      #angle axis calculation
      normal_vector = cross_product(touch1_pose_to_touch2_pose_if_no_rotation, touch1_pose_to_touch2_pose)
      normal_vector_norm = norm(normal_vector)
      if (normal_vector_norm > 10e-6):
        rotation_angle_rad = asin( normal_vector_norm / (norm(touch1_pose_to_touch2_pose_if_no_rotation) * norm(touch1_pose_to_touch2_pose) ) )
        normal_vector_to_angle_axis_multiply_norm_factor = rotation_angle_rad / normal_vector_norm
        angle_axis = [normal_vector[0] * normal_vector_to_angle_axis_multiply_norm_factor, normal_vector[1] * normal_vector_to_angle_axis_multiply_norm_factor, normal_vector[2] * normal_vector_to_angle_axis_multiply_norm_factor]
        rotation_offset_pose = p[0, 0, 0, angle_axis[0], angle_axis[1], angle_axis[2]]

        #rotate touch1 pose using touch2 information
        touch1_pose_rotated = pose_trans(touch1_pose, rotation_offset_pose)
      else:
        touch1_pose_rotated = touch1_pose
      end

      # relocate the feature using touch1_rotated_pose
      return relocate_xyzr(feature_init_pose, touch1_init_pose, touch1_pose_rotated)
    end

    def relocate_1_touch(touch_init_pose, touch_pose, feature_init_pose, feature_actual_pose):
      touch_initial_pose_in_initial_feature_frame = pose_trans(pose_inv(feature_init_pose), touch_init_pose)
      touch_actual_pose_in_actual_feature_frame = pose_trans(pose_inv(feature_actual_pose), touch_pose)

      # difference between touch poses in their respective feature frame
      touch_pose_offset = pose_sub(touch_actual_pose_in_actual_feature_frame, touch_initial_pose_in_initial_feature_frame)

      # remove all rotation from offset
      touch_pose_offset[3] = 0
      touch_pose_offset[4] = 0
      touch_pose_offset[5] = 0

      # apply pose offset to actual feature
      return pose_trans(feature_actual_pose, touch_pose_offset)
    end
    ##############################################
    # PALLETIZER INITIALIZATION
    ##############################################
    if(not palletizerXmlRpcClient.acknowledgePalletStates()):
      checkForScriptPreparationException()
      halt
    end

    ##############################################
    # PALLETIZER-RELATED VARIABLES AND METHODS
    ##############################################
    def rq_is_last_box_of_layer(box_id, end_of_layer_boxes):
      number_of_layers = length(end_of_layer_boxes)
      i = 0
      while i < number_of_layers:
        if box_id == end_of_layer_boxes[i]:
          return True
          break
        end
        i = i + 1
      end
      return False
    end

    def rq_is_palletOne_activated(pallet_one_current_box_count, pallet_two_current_box_count, second_pallet_activated):
      return ((pallet_one_current_box_count == 0) and (pallet_two_current_box_count == 0) and (not second_pallet_activated)) or (pallet_one_current_box_count > pallet_two_current_box_count)
    end
    global servojId = 2
  rq_collision_detection_stop()
  # end: URCap Installation Node
  # begin: URCap Installation Node
  #   Source: Robotiq_Grippers, 1.8.6.7016, Robotiq Inc.
  #   Type: Gripper
  rq_gripper_socket_ip_address = "127.0.0.1"
  rq_gripper_socket_port = 63352

  rq_comm_check_fail_counter = [0, 0, 0, 0]

  rq_read_act = [-1, -1, -1, -1]
  rq_read_gto = [-1, -1, -1, -1]
  rq_read_for = [-1, -1, -1, -1]
  rq_read_spe = [-1, -1, -1, -1]
  rq_read_obj = [-1, -1, -1, -1]
  rq_read_sta = [-1, -1, -1, -1]
  rq_read_flt = [-1, -1, -1, -1]
  rq_read_pos = [-1, -1, -1, -1]
  rq_read_pre = [-1, -1, -1, -1]
  rq_read_lbp = [-1, -1, -1, -1]
  rq_read_lrd = [-1, -1, -1, -1]
  rq_read_lbl = [-1, -1, -1, -1]
  rq_read_lgn = [-1, -1, -1, -1]
  rq_read_msc = [-1, -1, -1, -1]
  rq_read_mod = [-1, -1, -1, -1]
  rq_read_cou = [-1, -1, -1, -1]
  rq_read_ncy = [-1, -1, -1, -1]
  rq_read_dst = [-1, -1, -1, -1]
  rq_read_pco = [-1, -1, -1, -1]

  rq_string_initial_value = "N/A"

  rq_read_snu_1 = rq_string_initial_value
  rq_read_snu_2 = rq_string_initial_value
  rq_read_snu_3 = rq_string_initial_value
  rq_read_snu_4 = rq_string_initial_value

  rq_read_fwv_1 = rq_string_initial_value
  rq_read_fwv_2 = rq_string_initial_value
  rq_read_fwv_3 = rq_string_initial_value
  rq_read_fwv_4 = rq_string_initial_value

  rq_read_ver_1 = rq_string_initial_value
  rq_read_ver_2 = rq_string_initial_value
  rq_read_ver_3 = rq_string_initial_value
  rq_read_ver_4 = rq_string_initial_value

  rq_read_act_req = [True, True, True, True]
  rq_read_gto_req = [True, True, True, True]
  rq_read_for_req = [True, True, True, True]
  rq_read_spe_req = [True, True, True, True]
  rq_read_obj_req = [True, True, True, True]
  rq_read_sta_req = [True, True, True, True]
  rq_read_flt_req = [True, True, True, True]
  rq_read_pos_req = [True, True, True, True]
  rq_read_pre_req = [True, True, True, True]
  rq_read_lbp_req = [True, True, True, True]
  rq_read_lrd_req = [True, True, True, True]
  rq_read_lbl_req = [True, True, True, True]
  rq_read_lgn_req = [True, True, True, True]
  rq_read_msc_req = [True, True, True, True]
  rq_read_mod_req = [True, True, True, True]
  rq_read_cou_req = [True, True, True, True]
  rq_read_ncy_req = [True, True, True, True]
  rq_read_dst_req = [True, True, True, True]
  rq_read_pco_req = [True, True, True, True]

  rq_read_snu_1_req = False
  rq_read_snu_2_req = False
  rq_read_snu_3_req = False
  rq_read_snu_4_req = False

  rq_read_fwv_1_req = False
  rq_read_fwv_2_req = False
  rq_read_fwv_3_req = False
  rq_read_fwv_4_req = False

  rq_read_ver_1_req = False
  rq_read_ver_2_req = False
  rq_read_ver_3_req = False
  rq_read_ver_4_req = False

  rq_write_act_request = [False, False, False, False]
  rq_write_gto_request = [False, False, False, False]
  rq_write_atr_request = [False, False, False, False]
  rq_write_ard_request = [False, False, False, False]
  rq_write_pos_request = [False, False, False, False]
  rq_write_lbp_request = [False, False, False, False]
  rq_write_lrd_request = [False, False, False, False]
  rq_write_lbl_request = [False, False, False, False]
  rq_write_lgn_request = [False, False, False, False]
  rq_write_msc_request = [False, False, False, False]
  rq_write_mod_request = [False, False, False, False]

  rq_write_act = [-1, -1, -1, -1]
  rq_write_gto = [-1, -1, -1, -1]
  rq_write_atr = [-1, -1, -1, -1]
  rq_write_ard = [-1, -1, -1, -1]
  rq_write_for = [-1, -1, -1, -1]
  rq_write_spe = [-1, -1, -1, -1]
  rq_write_pos = [-1, -1, -1, -1]
  rq_write_lbp = [-1, -1, -1, -1]
  rq_write_lrd = [-1, -1, -1, -1]
  rq_write_lbl = [-1, -1, -1, -1]
  rq_write_lgn = [-1, -1, -1, -1]
  rq_write_msc = [-1, -1, -1, -1]
  rq_write_mod = [-1, -1, -1, -1]

  rq_write_act_previous = rq_write_act
  rq_write_gto_previous = rq_write_gto
  rq_write_atr_previous = rq_write_atr
  rq_write_ard_previous = rq_write_ard
  rq_write_for_previous = rq_write_for
  rq_write_spe_previous = rq_write_spe
  rq_write_pos_previous = rq_write_pos
  rq_write_lbp_previous = rq_write_lbp
  rq_write_lrd_previous = rq_write_lrd
  rq_write_lbl_previous = rq_write_lbl
  rq_write_lgn_previous = rq_write_lgn
  rq_write_msc_previous = rq_write_msc
  rq_write_mod_previous = rq_write_mod

  gripper_connected = [False, False, False, False]
  gripper_socket_open = [False, False, False, False]
  rq_comm_clear_socket_buffer_enabled = [True, True, True, True]
  rq_comm_check_counter = 0
  rq_gripper_communication_thread_started = False

  thread rq_gripper_communication():
      rq_comm_read_constants()
      rq_comm_read_variables()
      rq_comm_initialize_write_values()

      while(True):
          rq_comm_clear_socket_buffer()
          rq_comm_check()
          rq_comm_read_variables()
          rq_comm_write_variables()

          rq_gripper_communication_thread_started = True
          sleep(0.008)
      end
  end

  def rq_socket_to_index(gripper_socket="1"):
      # Patch in case gripper_socket is an integer
      gripper_socket_string = str_cat("", gripper_socket)

      if(gripper_socket_string == "1"):
          return 0
      elif(gripper_socket_string == "2"):
          return 1
      elif(gripper_socket_string == "3"):
          return 2
      elif(gripper_socket_string == "4"):
          return 3
      end
      return 0
  end

  def rq_index_to_socket(index=0):
      if(index == 0):
          return "1"
      elif(index == 1):
          return "2"
      elif(index == 2):
          return "3"
      elif(index == 3):
          return "4"
      end
      return "1"
  end

  def rq_comm_check():
      index = 0
      rq_comm_check_fail_counter_max = 99999

      if(rq_comm_check_counter < 50):
          rq_comm_check_counter = rq_comm_check_counter + 1
      else:
          rq_comm_check_counter = 0

          while(index <= 3):
              socket = rq_index_to_socket(index)

              if(gripper_connected[index]):
                  # Patch in case gripper_socket is an integer
                  gripper_socket_string = str_cat("", socket)

                  sid_list = rq_get_sid(socket)
                  is_gripper_in_sid_list = rq_is_gripper_in_sid_list(gripper_socket_string, sid_list)

                  if(is_gripper_in_sid_list):
                      rq_comm_check_fail_counter[index] = 0
                  else:
                      rq_comm_check_fail_counter[index] = rq_comm_check_fail_counter[index] + 1
                  end

                  if(rq_comm_check_fail_counter[index] > rq_comm_check_fail_counter_max):
                      message = str_cat("Communication lost with Robotiq's Gripper Slave ID ", gripper_socket_string)
                      popup(message, "Communication Error", False, True, True)
                  end
              end
              index = index + 1
          end
      end
  end

  def rq_init_comm_if_connected(gripper_sid=9, gripper_socket="1"):
      if(not is_gripper_socket_open(gripper_socket)):
        open_gripper_socket(gripper_socket)
      end

      socket_sid_set = rq_set_sid(gripper_sid, gripper_socket)

      if(socket_sid_set):
          # Patch in case gripper_socket is an integer
          gripper_socket_string = str_cat("", gripper_socket)

          sid_list = rq_get_sid(gripper_socket)
          is_gripper_in_sid_list = rq_is_gripper_in_sid_list(gripper_socket_string, sid_list)

          if(is_gripper_in_sid_list):
              rq_set_gripper_connected(gripper_socket_string)
              return True
          end
      end

      return False
  end

  def open_gripper_socket(gripper_socket="1"):
      is_open = socket_open(rq_gripper_socket_ip_address, rq_gripper_socket_port, gripper_socket)
      set_gripper_socket_open(gripper_socket, is_open)
  end

  def rq_close_gripper_socket(gripper_socket="1"):
      socket_close(gripper_socket)
      set_gripper_socket_open(gripper_socket, False)
      rq_set_gripper_connected(gripper_socket, False)
  end


  def is_gripper_socket_open(gripper_socket="1"):
      return gripper_socket_open[rq_socket_to_index(gripper_socket)]
  end

  def set_gripper_socket_open(gripper_socket, is_open):
      gripper_socket_open[rq_socket_to_index(gripper_socket)] = is_open
  end

  def rq_set_gripper_connected(gripper_socket="1", connected = True):
      gripper_connected[rq_socket_to_index(gripper_socket)] = connected
  end

  def rq_is_gripper_connected(gripper_id="1"):
      return gripper_connected[rq_socket_to_index(gripper_id)]
  end

  def rq_set_sid(gripper_sid=9, gripper_socket="1"):
      socket_set_var("SID", gripper_sid,  gripper_socket)
      ack = socket_read_byte_list(3, gripper_socket)
      return is_ack(ack)
  end

  def rq_get_sid(gripper_socket="1"):
      socket_send_string("GET SID", gripper_socket)
      sid_list = socket_read_byte_list(17, gripper_socket)
      return sid_list
  end

  def rq_wait_for_gripper_connected():
      gripper_socket = "gripper_conn_socket"
      socket_open(rq_gripper_socket_ip_address, rq_gripper_socket_port, gripper_socket)

      remainingRetries = 2000
      sid_list = rq_get_sid(gripper_socket)
      gripper_is_connected = rq_is_any_gripper_connected(sid_list)

      while(not gripper_is_connected and remainingRetries > 0):
          remainingRetries = remainingRetries - 1
          sid_list = rq_get_sid(gripper_socket)
          gripper_is_connected = rq_is_any_gripper_connected(sid_list)
      end

      socket_close(gripper_socket)
  end

  def rq_is_any_gripper_connected(sid_list):
      is_gripper_1_connected = rq_is_gripper1_in_sid_list(sid_list)
      is_gripper_2_connected = rq_is_gripper2_in_sid_list(sid_list)
      is_gripper_3_connected = rq_is_gripper3_in_sid_list(sid_list)
      is_gripper_4_connected = rq_is_gripper4_in_sid_list(sid_list)

      return is_gripper_1_connected or is_gripper_2_connected or is_gripper_3_connected or is_gripper_4_connected
  end

  def rq_is_gripper_ascii_in_sid_list(gripper_ascii_sid, sid_list):
      sid_list_length = sid_list[0]
      sid_list_empty_length = 2

      if (sid_list_length <= sid_list_empty_length):
          return False
      end

      sid1 = sid_list[2]
      sid2 = sid_list[5]
      sid3 = sid_list[8]
      sid4 = sid_list[11]

      return sid1 == gripper_ascii_sid or sid2 == gripper_ascii_sid or sid3 == gripper_ascii_sid or sid4 == gripper_ascii_sid
  end

  def rq_is_gripper_in_sid_list(gripper_socket_string, sid_list):
      if(gripper_socket_string == "1"):
          return rq_is_gripper1_in_sid_list(sid_list)
      elif(gripper_socket_string == "2"):
          return rq_is_gripper2_in_sid_list(sid_list)
      elif(gripper_socket_string == "3"):
          return rq_is_gripper3_in_sid_list(sid_list)
      elif(gripper_socket_string == "4"):
          return rq_is_gripper4_in_sid_list(sid_list)
      end
      return False
  end

  def rq_is_gripper1_in_sid_list(sid_list):
      gripper_1_sid_ascii = 57
      return rq_is_gripper_ascii_in_sid_list(gripper_1_sid_ascii, sid_list)
  end

  def rq_is_gripper2_in_sid_list(sid_list):
      gripper_2_sid_ascii = 50
      return rq_is_gripper_ascii_in_sid_list(gripper_2_sid_ascii, sid_list)
  end

  def rq_is_gripper3_in_sid_list(sid_list):
      gripper_3_sid_ascii = 51
      return rq_is_gripper_ascii_in_sid_list(gripper_3_sid_ascii, sid_list)
  end

  def rq_is_gripper4_in_sid_list(sid_list):
      gripper_4_sid_ascii = 52
      return rq_is_gripper_ascii_in_sid_list(gripper_4_sid_ascii, sid_list)
  end

  def rq_comm_clear_socket_buffer():
      index = 0

      while(index <= 3):
          socket = rq_index_to_socket(index)

          if(gripper_connected[index] and rq_comm_clear_socket_buffer_enabled[index]):
              byte_in_buffer = socket_read_byte_list(1, socket, 0.002)
              while(byte_in_buffer[0] >= 1):
                  byte_in_buffer = socket_read_byte_list(1, socket, 0.002)
              end
              rq_comm_clear_socket_buffer_enabled[index] = False
          end
          index = index + 1
      end
  end

  def rq_comm_initialize_write_values():
      index = 0

      while(index <= 3):
          socket = rq_index_to_socket(index)

          if(gripper_connected[index]):

              if(rq_write_act[index] == -1 and rq_read_act[index] != -1):
                  rq_write_act[index] = rq_read_act[index]
                  rq_write_act_previous[index] = rq_read_act[index]
              elif(rq_write_act_previous[index] == -1 and rq_read_act[index] != -1):
                  rq_write_act_previous[index] = rq_read_act[index]
              end

              if(rq_write_gto[index] == -1 and rq_read_gto[index] != -1):
                  rq_write_gto[index] = rq_read_gto[index]
                  rq_write_gto_previous[index] = rq_read_gto[index]
              elif(rq_write_gto_previous[index] == -1 and rq_read_gto[index] != -1):
                  rq_write_gto_previous[index] = rq_read_gto[index]
              end

              if(rq_write_for[index] == -1 and rq_read_for[index] != -1):
                  rq_write_for[index] = rq_read_for[index]
                  rq_write_for_previous[index] = rq_read_for[index]
              elif(rq_write_for_previous[index] == -1 and rq_read_for[index] != -1):
                  rq_write_for_previous[index] = rq_read_for[index]
              end

              if(rq_write_spe[index] == -1 and rq_read_spe[index] != -1):
                  rq_write_spe[index] = rq_read_spe[index]
                  rq_write_spe_previous[index] = rq_read_spe[index]
              elif(rq_write_spe_previous[index] == -1 and rq_read_spe[index] != -1):
                  rq_write_spe_previous[index] = rq_read_spe[index]
              end

              if(rq_write_pos[index] == -1 and rq_read_pos[index] != -1):
                  rq_write_pos[index] = rq_read_pos[index]
                  rq_write_pos_previous[index] = rq_read_pos[index]
              elif(rq_write_pos_previous[index] == -1 and rq_read_pos[index] != -1):
                  rq_write_pos_previous[index] = rq_read_pos[index]
              end

              if(rq_write_lbp[index] == -1 and rq_read_lbp[index] != -1):
                  rq_write_lbp[index] = rq_read_lbp[index]
                  rq_write_lbp_previous[index] = rq_read_lbp[index]
              elif(rq_write_lbp_previous[index] == -1 and rq_read_lbp[index] != -1):
                  rq_write_lbp_previous[index] = rq_read_lbp[index]
              end

              if(rq_write_lrd[index] == -1 and rq_read_lrd[index] != -1):
                  rq_write_lrd[index] = rq_read_lrd[index]
                  rq_write_lrd_previous[index] = rq_read_lrd[index]
              elif(rq_write_lrd_previous[index] == -1 and rq_read_lrd[index] != -1):
                  rq_write_lrd_previous[index] = rq_read_lrd[index]
              end

              if(rq_write_lbl[index] == -1 and rq_read_lbl[index] != -1):
                  rq_write_lbl[index] = rq_read_lbl[index]
                  rq_write_lbl_previous[index] = rq_read_lbl[index]
              elif(rq_write_lbl_previous[index] == -1 and rq_read_lbl[index] != -1):
                  rq_write_lbl_previous[index] = rq_read_lbl[index]
              end

              if(rq_write_lgn[index] == -1 and rq_read_lgn[index] != -1):
                  rq_write_lgn[index] = rq_read_lgn[index]
                  rq_write_lgn_previous[index] = rq_read_lgn[index]
              elif(rq_write_lgn_previous[index] == -1 and rq_read_lgn[index] != -1):
                  rq_write_lgn_previous[index] = rq_read_lgn[index]
              end

              if(rq_write_msc[index] == -1 and rq_read_msc[index] != -1):
                  rq_write_msc[index] = rq_read_msc[index]
                  rq_write_msc_previous[index] = rq_read_msc[index]
              elif(rq_write_msc_previous[index] == -1 and rq_read_msc[index] != -1):
                  rq_write_msc_previous[index] = rq_read_msc[index]
              end

              if(rq_write_mod[index] == -1 and rq_read_mod[index] != -1):
                  rq_write_mod[index] = rq_read_mod[index]
                  rq_write_mod_previous[index] = rq_read_mod[index]
              elif(rq_write_mod_previous[index] == -1 and rq_read_mod[index] != -1):
                  rq_write_mod_previous[index] = rq_read_mod[index]
              end

          end
          index = index + 1
      end
  end

  def rq_comm_set_var(var, value=0, gripper_socket="1"):
      socket_set_var(var, value, gripper_socket)
      return socket_read_byte_list(3, gripper_socket)
  end

  def rq_comm_set_pos_spe_for(pos=0, speed=0, force=0, gripper_socket="1"):
      socket_send_string("SET POS", gripper_socket)
      socket_send_byte(32, gripper_socket)
      socket_send_string(pos, gripper_socket)
      socket_send_byte(32, gripper_socket)
      socket_send_string("SPE", gripper_socket)
      socket_send_byte(32, gripper_socket)
      socket_send_string(speed, gripper_socket)
      socket_send_byte(32, gripper_socket)
      socket_send_string("FOR", gripper_socket)
      socket_send_byte(32, gripper_socket)
      socket_send_string(force, gripper_socket)
      socket_send_byte(10, gripper_socket)
      return socket_read_byte_list(3, gripper_socket)
  end

  def rq_comm_read_variables():
      index = 0

      while(index <= 3):
          socket = rq_index_to_socket(index)

          if(gripper_connected[index]):

              if(rq_read_act_req[index]):
                  rq_read_act[index] = socket_get_var("ACT", socket)
                  rq_read_act_req[index] = False
              end

              if(rq_read_gto_req[index]):
                  rq_read_gto[index] = socket_get_var("GTO", socket)
                  rq_read_gto_req[index] = False
              end

              if(rq_read_pre_req[index]):
                  rq_read_pre[index] = socket_get_var("PRE", socket)
                  rq_read_pre_req[index] = False
              end

              if(rq_read_pos_req[index]):
                  rq_read_pos[index] = socket_get_var("POS", socket)
                  rq_read_pos_req[index] = False
              end

              if(rq_read_spe_req[index]):
                  rq_read_spe[index] = socket_get_var("SPE", socket)
                  rq_read_spe_req[index] = False
              end

              if(rq_read_for_req[index]):
                  rq_read_for[index] = socket_get_var("FOR", socket)
                  rq_read_for_req[index] = False
              end

              if(rq_read_obj_req[index]):
                  rq_read_obj[index] = socket_get_var("OBJ", socket)
                  rq_read_obj_req[index] = False
              end

              if(rq_read_sta_req[index]):
                  rq_read_sta[index] = socket_get_var("STA", socket)
                  rq_read_sta_req[index] = False
              end

              if(rq_read_mod_req[index]):
                  rq_read_mod[index] = socket_get_var("MOD", socket)
                  rq_read_mod_req[index] = False
              end

              if(rq_read_flt_req[index]):
                  rq_read_flt[index] = socket_get_var("FLT",socket)
                  rq_read_flt_req[index] = False
              end

              if(rq_read_lbp_req[index]):
                  rq_read_lbp[index] = socket_get_var("LBP", socket)
                  rq_read_lbp_req[index] = False
              end

              if(rq_read_lrd_req[index]):
                  rq_read_lrd[index] = socket_get_var("LRD", socket)
                  rq_read_lrd_req[index] = False
              end

              if(rq_read_lbl_req[index]):
                  rq_read_lbl[index] = socket_get_var("LBL",socket)
                  rq_read_lbl_req[index] = False
              end

              if(rq_read_lgn_req[index]):
                  rq_read_lgn[index] = socket_get_var("LGN", socket)
                  rq_read_lgn_req[index] = False
              end

              if(rq_read_msc_req[index]):
                  rq_read_msc[index] = socket_get_var("MSC", socket)
                  rq_read_msc_req[index] = False
              end

              if(rq_read_cou_req[index]):
                  rq_read_cou[index] = socket_get_var("COU", socket)
                  rq_read_cou_req[index] = False
              end

              if(rq_read_ncy_req[index]):
                  rq_read_ncy[index] = socket_get_var("NCY", socket)
                  rq_read_ncy_req[index] = False
              end

              if(rq_read_dst_req[index]):
                  rq_read_dst[index] = socket_get_var("DST", socket)
                  rq_read_dst_req[index] = False
              end

              if(rq_read_pco_req[index]):
                  rq_read_pco[index] = socket_get_var("PCO", socket)
                  rq_read_pco_req[index] = False
              end
          end
          index = index + 1
      end
  end

  def rq_comm_read_constants():

      if(gripper_connected[0]):
          while(rq_read_snu_1 == rq_string_initial_value):
              socket_send_string("GET SNU", "1")
              rq_read_snu_1 = socket_read_string("1")
          end

          while(rq_read_fwv_1 == rq_string_initial_value):
              socket_send_string("GET FWV", "1")
              rq_read_fwv_1 = socket_read_string("1")
          end

          while(rq_read_ver_1 == rq_string_initial_value):
              socket_send_string("GET VER", "1")
              rq_read_ver_1 = socket_read_string("1")
          end
      end

      if(gripper_connected[1]):
          while(rq_read_snu_2 == rq_string_initial_value):
              socket_send_string("GET SNU", "2")
              rq_read_snu_2 = socket_read_string("2")
          end

          while(rq_read_fwv_2 == rq_string_initial_value):
              socket_send_string("GET FWV", "2")
              rq_read_fwv_2 = socket_read_string("2")
          end

          while(rq_read_ver_2 == rq_string_initial_value):
              socket_send_string("GET VER", "2")
              rq_read_ver_2 = socket_read_string("2")
          end
      end

      if(gripper_connected[2]):
          while(rq_read_snu_3 == rq_string_initial_value):
              socket_send_string("GET SNU", "3")
              rq_read_snu_3 = socket_read_string("3")
          end

          while(rq_read_fwv_3 == rq_string_initial_value):
              socket_send_string("GET FWV", "3")
              rq_read_fwv_3 = socket_read_string("3")
          end

          while(rq_read_ver_3 == rq_string_initial_value):
              socket_send_string("GET VER", "3")
              rq_read_ver_3 = socket_read_string("3")
          end
      end

      if(gripper_connected[3]):
          while(rq_read_snu_4 == rq_string_initial_value):
              socket_send_string("GET SNU", "4")
              rq_read_snu_4 = socket_read_string("4")
          end

          while(rq_read_fwv_4 == rq_string_initial_value):
              socket_send_string("GET FWV", "4")
              rq_read_fwv_4 = socket_read_string("4")
          end

          while(rq_read_ver_4 == rq_string_initial_value):
              socket_send_string("GET VER", "4")
              rq_read_ver_4 = socket_read_string("4")
          end
      end
  end

  def rq_comm_write_variables():
      index = 0

      while(index <= 3):
          socket = rq_index_to_socket(index)

          if(gripper_connected[index]):

              if(rq_write_act_request[index]):
                  if(is_ack(rq_comm_set_var("ACT", rq_write_act[index], socket))):
                      rq_write_act_previous[index] = rq_write_act[index]
                      rq_write_act_request[index] = False
                  end
              end

              if(rq_write_gto_request[index]):
                  if(is_ack(rq_comm_set_var("GTO", rq_write_gto[index], socket))):
                      rq_write_gto_previous[index] = rq_write_gto[index]
                      rq_write_gto_request[index] = False
                  end
              end

              if(rq_write_atr_request[index]):
                  if(is_ack(rq_comm_set_var("ATR", rq_write_atr[index], socket))):
                      rq_write_atr_previous[index] = rq_write_atr[index]
                      rq_write_atr_request[index] = False
                  end
              end

              if(rq_write_ard_request[index]):
                  if(is_ack(rq_comm_set_var("ARD", rq_write_ard[index], socket))):
                      rq_write_ard_previous[index] = rq_write_ard[index]
                      rq_write_ard_request[index] = False
                  end
              end

              if(rq_write_pos_request[index]):
                  if(is_ack(rq_comm_set_pos_spe_for(rq_write_pos[index], rq_write_spe[index], rq_write_for[index], socket))):
                      rq_write_pos_previous[index] = rq_write_pos[index]
                      rq_write_spe_previous[index] = rq_write_spe[index]
                      rq_write_for_previous[index] = rq_write_for[index]
                      rq_write_pos_request[index] = False
                  end
              end

              if(rq_write_lbp_request[index]):
                  if(is_ack(rq_comm_set_var("LBP", rq_write_lbp[index], socket))):
                      rq_write_lbp_previous[index] = rq_write_lbp[index]
                      rq_write_lbp_request[index] = False
                  end
              end

              if(rq_write_lrd_request[index]):
                  if(is_ack(rq_comm_set_var("LRD", rq_write_lrd[index], socket))):
                      rq_write_lrd_previous[index] = rq_write_lrd[index]
                      rq_write_lrd_request[index] = False
                  end
              end

              if(rq_write_lbl_request[index]):
                  if(is_ack(rq_comm_set_var("LBL", rq_write_lbl[index], socket))):
                      rq_write_lbl_previous[index] = rq_write_lbl[index]
                      rq_write_lbl_request[index] = False
                  end
              end

              if(rq_write_lgn_request[index]):
                  if(is_ack(rq_comm_set_var("LGN", rq_write_lgn[index], socket))):
                      rq_write_lgn_previous[index] = rq_write_lgn[index]
                      rq_write_lgn_request[index] = False
                  end
              end

              if(rq_write_msc_request[index]):
                  if(is_ack(rq_comm_set_var("MSC", rq_write_msc[index], socket))):
                      rq_write_msc_previous[index] = rq_write_msc[index]
                      rq_write_msc_request[index] = False
                  end
              end

              if(rq_write_mod_request[index]):
                  if(is_ack(rq_comm_set_var("MOD", rq_write_mod[index], socket))):
                      rq_write_mod_previous[index] = rq_write_mod[index]
                      rq_write_mod_request[index] = False
                  end
              end
          end
          index = index + 1
      end
  end

  def rq_activate(gripper_socket="1"):
      if (not rq_is_gripper_activated(gripper_socket)):
          rq_reset(gripper_socket)

          while(not rq_get_var("ACT", 1, gripper_socket) == 0 or not rq_get_var("STA", 1, gripper_socket) == 0):
              rq_reset(gripper_socket)
              sleep(0.008)
          end

          rq_set_var("ACT",1, gripper_socket)
      end
  end

  def rq_activate_and_wait(gripper_socket="1"):
      if (not rq_is_gripper_activated(gripper_socket)):
          rq_activate(gripper_socket)
          sleep(1.0)

          while(not rq_get_var("ACT", 1, gripper_socket) == 1 or not rq_get_var("STA", 1, gripper_socket) == 3):
              sleep(0.1)
          end

          sleep(0.5)
      end
  end

  def rq_activate_all_grippers(reset=False):
      if(gripper_connected[0]):
          rq_reset_and_activate("1", reset)
      end

      if(gripper_connected[1]):
          rq_reset_and_activate("2", reset)
      end

      if(gripper_connected[2]):
          rq_reset_and_activate("3", reset)
      end

      if(gripper_connected[3]):
          rq_reset_and_activate("4", reset)
      end
  end

  def rq_reset_and_activate(gripper_socket="1", reset=False):
      if(reset):
          rq_reset(gripper_socket)
          rq_activate_and_wait(gripper_socket)
      elif(not rq_is_gripper_activated(gripper_socket)):
          rq_activate_and_wait(gripper_socket)
      end
  end

  def rq_reset(gripper_socket="1"):
      rq_set_var("ACT", 0, gripper_socket)
      rq_set_var("ATR", 0, gripper_socket)

      while(not rq_get_var("ACT", 1, gripper_socket) == 0 or not rq_get_var("STA", 1, gripper_socket) == 0):
          rq_set_var("ACT", 0, gripper_socket)
          rq_set_var("ATR", 0, gripper_socket)
          sleep(0.008)
      end

      sleep(0.5)
  end

  def rq_auto_release_open_and_wait(gripper_socket="1"):
      rq_set_var("ATR",0, gripper_socket)
      rq_set_var("ARD",0, gripper_socket)
      rq_set_var("ACT",1, gripper_socket)
      sleep(0.1)
      rq_set_var("ATR",1, gripper_socket)

      rq_wait_autorelease_completed(gripper_socket)
  end

  def rq_auto_release_close_and_wait(gripper_socket="1"):
      rq_set_var("ATR",0, gripper_socket)
      rq_set_var("ARD",1, gripper_socket)
      rq_set_var("ACT",1, gripper_socket)
      sleep(0.1)
      rq_set_var("ATR",1, gripper_socket)

      rq_wait_autorelease_completed(gripper_socket)
  end

  def rq_wait_autorelease_completed(gripper_socket="1"):
      remainingRetries = 20
      gFLT = rq_get_var("FLT", 2, gripper_socket)

      while(not is_FLT_autorelease_in_progress(gFLT) and remainingRetries > 0):
          remainingRetries = remainingRetries - 1
          gFLT = rq_get_var("FLT", 2, gripper_socket)
          sleep(0.1)
      end

      remainingRetries = 100
      gFLT = rq_get_var("FLT", 2, gripper_socket)

      while(not is_FLT_autorelease_completed(gFLT) and remainingRetries > 0):
          remainingRetries = remainingRetries - 1
          gFLT = rq_get_var("FLT", 2, gripper_socket)
          sleep(0.1)
      end
  end

  def rq_set_force(force, gripper_socket="1"):
      force = floor(scale(force, [0, 255], [0.0, 255.0]))
      rq_set_var("FOR", force, gripper_socket)
  end

  def rq_set_speed(speed, gripper_socket="1"):
      speed = floor(scale(speed, [0, 255], [0.0, 255.0]))
      rq_set_var("SPE", speed, gripper_socket)
  end

  def rq_open(gripper_socket="1"):
      rq_move(0, gripper_socket)
  end

  def rq_close(gripper_socket="1"):
      rq_move(255, gripper_socket)
  end

  def rq_open_and_wait(gripper_socket="1"):
      rq_move_and_wait(0, gripper_socket)
  end

  def rq_close_and_wait(gripper_socket="1"):
      rq_move_and_wait(255, gripper_socket)
  end

  def rq_move(pos, gripper_socket="1"):
      rq_set_pos(pos, gripper_socket)
      rq_go_to(gripper_socket)
  end

  def rq_move_and_wait(pos, gripper_socket="1"):
      rq_move(pos, gripper_socket)

      while (not rq_is_motion_complete(gripper_socket)):
          # wait for motion completed
          sleep(0.008)
      end
  end

  def rq_wait_for_pos_request(pos, gripper_socket="1"):
      gPRE = rq_get_var("PRE", 3, gripper_socket)

      while (gPRE != pos):
          rq_set_var("POS", pos, gripper_socket)
          sleep(0.008)
          gPRE = rq_get_var("PRE", 3, gripper_socket)
      end
  end

  def rq_wait_pos_spe_for_request(pos, speed, force, gripper_socket="1"):
      gPRE = rq_get_var("PRE", 3, gripper_socket)

      while (gPRE != pos):
          rq_set_pos_spe_for_var(pos, speed, force, gripper_socket)
          sleep(0.008)
          gPRE = rq_get_var("PRE", 3, gripper_socket)
      end
  end

  def rq_wait_for_pos(pos, gripper_socket="1"):
      rq_wait_for_pos_request(pos, gripper_socket)

      # Wait for the gripper motion to complete
      while (not rq_is_motion_complete(gripper_socket)):
          # wait for motion completed
          sleep(0.008)
          rq_set_var("GTO", 1, gripper_socket)
      end
  end

  def rq_wait(gripper_socket="1"):
      # Wait for the gripper motion to complete
      while (not rq_is_motion_complete(gripper_socket)):
          sleep(0.008)
          # The following patch is for Robotiq's Camera issue when communication is lost, but not the activation
          # the communication driver reset the GTO bit
          rq_set_var("GTO", 1, gripper_socket)
      end
  end

  def rq_wait_for_object_detected(gripper_socket="1"):
      # Wait the object detection
      while (not rq_is_object_detected(gripper_socket)):
          sleep(0.008)
      end
  end

  # set the position
  def rq_set_pos(pos, gripper_socket="1"):
      pos = floor(scale(pos, [0, 255], [0.0, 255.0]))
      rq_set_var("POS", pos, gripper_socket)
      rq_wait_for_pos_request(pos, gripper_socket)
  end

  def rq_set_pos_spd_for(pos, speed, force, gripper_socket="1"):
      pos = floor(scale(pos, [0, 255], [0.0, 255.0]))
      speed = floor(scale(speed, [0, 255], [0.0, 255.0]))
      force = floor(scale(force, [0, 255], [0.0, 255.0]))

      rq_set_pos_spe_for_var(pos, speed, force, gripper_socket)
  end

  def rq_set_gripper_max_current_mA(current_mA, gripper_socket="1"):
      current = floor(current_mA / 10)

      rq_set_var("MSC", current, gripper_socket)
      current_read = rq_get_var("MSC", 1, gripper_socket)

      while(current_read != current):
          rq_set_var("MSC", current, gripper_socket)
          current_read = rq_get_var("MSC", 1, gripper_socket)
      end
  end

  def rq_set_gripper_mode(mode, gripper_socket="1"):
      rq_set_var("MOD", mode, gripper_socket)
  end

  def rq_set_gripper_max_cur(current_mA, gripper_socket="1"):
      rq_set_gripper_max_current_mA(current_mA, gripper_socket)
  end

  def rq_get_gripper_max_current_mA(gripper_socket="1"):
      current = rq_get_var("MSC", 1, gripper_socket)

      if(current == -1):
          current_mA = current
      else:
          current_mA = current * 10
      end

      return current_mA
  end

  def rq_get_gripper_max_cur(gripper_socket="1"):
      return rq_get_gripper_max_current_mA(gripper_socket)
  end

  def rq_set_max_current_for_all_grippers():
      current_mA = rq_get_max_current_mA()

      if(gripper_connected[0]):
          rq_set_gripper_max_current_mA(current_mA, "1")
      end

      if(gripper_connected[1]):
          rq_set_gripper_max_current_mA(current_mA, "2")
      end

      if(gripper_connected[2]):
          rq_set_gripper_max_current_mA(current_mA, "3")
      end

      if(gripper_connected[3]):
          rq_set_gripper_max_current_mA(current_mA, "4")
      end
  end

  def rq_get_max_current_mA():
      max_current_mA = 0

      if(rq_current_limit_enabled):
          nb_connected_grippers = rq_get_nb_connected_grippers()

          if(nb_connected_grippers == 1):
              max_current_mA = 600
          elif(nb_connected_grippers > 1):
              max_current_mA = 450
          end
      else:

      end

      return max_current_mA
  end

  def rq_get_nb_connected_grippers():
      nb_connected_grippers = 0

      if(gripper_connected[0]):
          nb_connected_grippers = nb_connected_grippers + 1
      end

      if(gripper_connected[1]):
          nb_connected_grippers = nb_connected_grippers + 1
      end

      if(gripper_connected[2]):
          nb_connected_grippers = nb_connected_grippers + 1
      end

      if(gripper_connected[3]):
          nb_connected_grippers = nb_connected_grippers + 1
      end

      return nb_connected_grippers
  end

  def rq_list_of_bytes_to_value(list_of_bytes):
      value = -1

      # response list length
      if (list_of_bytes[0] == 1):
          value = list_of_bytes[1] - 48
      elif (list_of_bytes[0] == 2):
          value = (list_of_bytes[1] - 48) * 10 + (list_of_bytes[2] - 48)
      elif (list_of_bytes[0] == 3):
          value = (list_of_bytes[1] - 48) * 100 + (list_of_bytes[2] - 48) * 10 + (list_of_bytes[3] - 48)
      end

      return value
  end

  def rq_is_motion_complete(gripper_socket="1"):
      gOBJ = rq_get_var("OBJ", 1, gripper_socket)
      sleep(0.008)
      return is_OBJ_gripper_at_position(gOBJ) or is_OBJ_object_detected(gOBJ)
  end

  def rq_is_gripper_activated(gripper_socket="1"):
      gSTA = rq_get_var("STA", 1, gripper_socket)
      sleep(0.008)
      return is_STA_gripper_activated(gSTA)
  end

  def rq_is_object_detected(gripper_socket="1"):
      gOBJ = rq_get_var("OBJ", 1, gripper_socket)
      sleep(0.008)
      return is_OBJ_object_detected(gOBJ)
  end

  def rq_current_pos(gripper_socket="1"):
      gPOS = rq_get_var("POS", 1, gripper_socket)
      sleep(0.008)
      return gPOS
  end

  def rq_motor_current(gripper_socket="1"):
      rq_current = rq_get_var("COU", 1, gripper_socket)
      sleep(0.008)
      return rq_current * 10
  end

  def rq_print_connected_grippers():
      if(gripper_connected[0]):
          textmsg("Gripper 1 : ", "connected and socket open.")
      end

      if (gripper_connected[1]):
          textmsg("Gripper 2 : ", "connected and socket open.")
      end

      if (gripper_connected[2]):
          textmsg("Gripper 3 : ", "connected and socket open.")
      end

      if (gripper_connected[3]):
          textmsg("Gripper 4 : ", "connected and socket open.")
      end
  end

  def rq_print_gripper_fault_code(gripper_socket="1"):
      gFLT = rq_get_var("FLT", 2, gripper_socket)

      if(is_FLT_no_fault(gFLT)):
          textmsg("Gripper Fault : ", "No Fault (0x00)")
      elif (is_FLT_action_delayed(gFLT)):
          textmsg("Gripper Fault : ", "Priority Fault: Action delayed, initialization must be completed prior to action (0x05)")
      elif (is_FLT_not_activated(gFLT)):
          textmsg("Gripper Fault : ", "Priority Fault: The activation must be set prior to action (0x07)")
      elif (is_FLT_autorelease_in_progress(gFLT)):
          textmsg("Gripper Fault : ", "Minor Fault: Automatic release in progress (0x0B)")
      elif (is_FLT_overcurrent(gFLT)):
          textmsg("Gripper Fault : ", "Minor Fault: Overcurrent protection triggered (0x0E)")
      elif (is_FLT_autorelease_completed(gFLT)):
          textmsg("Gripper Fault : ", "Major Fault: Automatic release completed (0x0F)")
      else:
          textmsg("Gripper Fault : ", "Unknown Fault")
      end
  end

  def rq_print_gripper_num_cycles(gripper_socket="1"):
      num_cycles = rq_get_var("NCY", 1, gripper_socket)

      if(num_cycles == -1):
          textmsg("Gripper Cycle Number : ", "Number of cycles is unreachable.")
      else:
          textmsg("Gripper Cycle Number : ", num_cycles)
      end
  end

  def rq_print_gripper_driver_state(gripper_socket="1"):
      driver_state = rq_get_var("DST", 1, gripper_socket)

      if(driver_state == 0):
          textmsg("Gripper Driver State : ", "RQ_STATE_INIT")
      elif(driver_state == 1):
          textmsg("Gripper Driver State : ", "RQ_STATE_LISTEN")
      elif(driver_state == 2):
          textmsg("Gripper Driver State : ", "RQ_STATE_READ_INFO")
      elif(driver_state == 3):
          textmsg("Gripper Driver State : ", "RQ_STATE_ACTIVATION")
      else:
          textmsg("Gripper Driver State : ", "RQ_STATE_RUN")
      end
  end

  def rq_print_gripper_serial_number(gripper_socket="1"):
      serial_number = rq_get_var_string("SNU", 1, gripper_socket)
      textmsg("Gripper Serial Number : ", serial_number)
  end

  def rq_print_gripper_firmware_version(gripper_socket="1"):
      firmware_version = rq_get_var_string("FWV", 1, gripper_socket)
      textmsg("Gripper Firmware Version : ", firmware_version)
  end

  def rq_print_gripper_driver_version(gripper_socket="1"):
      driver_version = rq_get_var_string("VER", 1, gripper_socket)
      textmsg("Gripper Driver Version : ", driver_version)
  end

  def rq_print_gripper_connection_state(gripper_socket="1"):
      connection_state = rq_get_var("PCO", 1, gripper_socket)

      if (connection_state == 0):
          textmsg("Gripper Connection State : ", "No connection problem detected")
      else:
          textmsg("Gripper Connection State : ", "Connection problem detected")
      end
  end

  # Returns True if list_of_bytes is [3, 'a', 'c', 'k']
  def is_ack(list_of_bytes):

      # list length is not 3
      if (list_of_bytes[0] != 3):
          return False
      end

      # first byte not is 'a'?
      if (list_of_bytes[1] != 97):
          return False
      end

      # first byte not is 'c'?
      if (list_of_bytes[2] != 99):
          return False
      end

      # first byte not is 'k'?
      if (list_of_bytes[3] != 107):
          return False
      end

      return True
  end

  # Returns True if list_of_bytes is not [3, 'a', 'c', 'k']
  def is_not_ack(list_of_bytes):
      if (is_ack(list_of_bytes)):
          return False
      else:
          return True
      end
  end

  def is_STA_gripper_activated (gSTA):
      if (gSTA == 3):
          return True
      end

      return False
  end

  def is_OBJ_object_detected (gOBJ):
      if (gOBJ == 1 or gOBJ == 2):
          return True
      end

      return False
  end

  def is_OBJ_gripper_at_position (gOBJ):
      if (gOBJ == 3):
          return True
      end

      return False
  end

  def is_not_OBJ_gripper_at_position (gOBJ):
      if (is_OBJ_gripper_at_position(gOBJ)):
          return False
      else:
          return True
      end
  end

  #### GTO Section ####
  def rq_stop(gripper_socket="1"):
      rq_set_var("GTO", 0, gripper_socket)
  end

  def rq_set_GTO_and_wait(value, gripper_socket="1"):
      rq_set_var("GTO" ,value, gripper_socket)
      while(not is_GTO(value, rq_get_var("GTO", 1, gripper_socket))):
        sleep(0.008)
      end
  end

  def rq_go_to(gripper_socket="1"):
      rq_set_var("GTO", 1, gripper_socket)
  end


  def is_GTO(goto_value, rGTO):
      return rGTO == goto_value
  end
  #### GTO Section ####

  def is_FLT_no_fault(gFLT):
      return gFLT == 0
  end

  def is_FLT_warning(gFLT):
      return gFLT >= 1 and gFLT <= 7
  end

  def is_FLT_faulted(gFLT):
      return gFLT >= 8
  end

  def is_FLT_action_delayed(gFLT):
      return gFLT == 5
  end

  def is_FLT_not_activated(gFLT):
      return gFLT == 7
  end

  def is_FLT_autorelease_in_progress(gFLT):
      return gFLT == 11
  end

  def is_FLT_overcurrent(gFLT):
      return gFLT == 14
  end

  def is_FLT_autorelease_completed(gFLT):
      return gFLT == 15
  end

  def rq_set_var(var_name, var_value, gripper_socket="1"):
      index = rq_socket_to_index(gripper_socket)

      enter_critical

      if (var_name == "ACT"):
          rq_write_act[index] = var_value
          rq_write_act_request[index] = True
      elif (var_name == "GTO"):
          rq_write_gto[index] = var_value
          rq_write_gto_request[index] = True
      elif (var_name == "ATR"):
          rq_write_atr[index] = var_value
          rq_write_atr_request[index] = True
      elif (var_name == "ARD"):
          rq_write_ard[index] = var_value
          rq_write_ard_request[index] = True
      elif (var_name == "FOR"):
          rq_write_for[index] = var_value
          rq_write_pos_request[index] = True
      elif (var_name == "SPE"):
          rq_write_spe[index] = var_value
          rq_write_pos_request[index] = True
      elif (var_name == "POS"):
          rq_write_pos[index] = var_value
          rq_write_pos_request[index] = True
      elif (var_name == "LBP"):
          rq_write_lbp[index] = var_value
          rq_write_lbp_request[index] = True
      elif (var_name == "LRD"):
          rq_write_lrd[index] = var_value
          rq_write_lrd_request[index] = True
      elif (var_name == "LBL"):
          rq_write_lbl[index] = var_value
          rq_write_lbl_request[index] = True
      elif (var_name == "LGN"):
          rq_write_lgn[index] = var_value
          rq_write_lgn_request[index] = True
      elif (var_name == "MSC"):
          rq_write_msc[index] = var_value
          rq_write_msc_request[index] = True
      elif (var_name == "MOD"):
          rq_write_mod[index] = var_value
          rq_write_mod_request[index] = True
      end

      exit_critical

      if (var_name == "ACT"):
          while(rq_write_act_request[index]):
              sleep(0.008)
          end
      elif (var_name == "GTO"):
          while(rq_write_gto_request[index]):
              sleep(0.008)
          end
      elif (var_name == "ATR"):
          while(rq_write_atr_request[index]):
              sleep(0.008)
          end
      elif (var_name == "ARD"):
          while(rq_write_ard_request[index]):
              sleep(0.008)
          end
      elif (var_name == "FOR"):
          while(rq_write_pos_request[index]):
              sleep(0.008)
          end
      elif (var_name == "SPE"):
          while(rq_write_pos_request[index]):
              sleep(0.008)
          end
      elif (var_name == "POS"):
          while(rq_write_pos_request[index]):
              sleep(0.008)
          end
      elif (var_name == "LBP"):
          while(rq_write_lbp_request[index]):
              sleep(0.008)
          end
      elif (var_name == "LRD"):
          while(rq_write_lrd_request[index]):
              sleep(0.008)
          end
      elif (var_name == "LBL"):
          while(rq_write_lbl_request[index]):
              sleep(0.008)
          end
      elif (var_name == "LGN"):
          while(rq_write_lgn_request[index]):
              sleep(0.008)
          end
      elif (var_name == "MSC"):
          while(rq_write_msc_request[index]):
              sleep(0.008)
          end
      elif (var_name == "MOD"):
          while(rq_write_mod_request[index]):
              sleep(0.008)
          end
      end
  end

  def rq_set_pos_spe_for_var(pos, speed, force, gripper_socket="1"):
      index = rq_socket_to_index(gripper_socket)

      enter_critical

      rq_write_for[index] = force
      rq_write_spe[index] = speed
      rq_write_pos[index] = pos
      rq_write_pos_request[index] = True

      exit_critical
  end

  def rq_get_var(var_name, nbr_bytes, gripper_socket="1"):
      index = rq_socket_to_index(gripper_socket)
      var_value = -1

      if (var_name == "ACT"):
          enter_critical
          rq_read_act_req[index] = True
          exit_critical
          while(rq_read_act_req[index]):
              sleep(0.008)
          end
          var_value = rq_read_act[index]

      elif (var_name == "GTO"):
          enter_critical
          rq_read_gto_req[index] = True
          exit_critical
          while(rq_read_gto_req[index]):
              sleep(0.008)
          end
          var_value = rq_read_gto[index]

      elif (var_name == "FOR"):
          enter_critical
          rq_read_for_req[index] = True
          exit_critical
          while(rq_read_for_req[index]):
              sleep(0.008)
          end
          var_value = rq_read_for[index]

      elif (var_name == "SPE"):
          enter_critical
          rq_read_spe_req[index] = True
          exit_critical
          while(rq_read_spe_req[index]):
              sleep(0.008)
          end
          var_value = rq_read_spe[index]

      elif (var_name == "OBJ"):
          enter_critical
          rq_read_obj_req[index] = True
          exit_critical
          while(rq_read_obj_req[index]):
              sleep(0.008)
          end
          var_value = rq_read_obj[index]

      elif (var_name == "STA"):
          enter_critical
          rq_read_sta_req[index] = True
          exit_critical
          while(rq_read_sta_req[index]):
              sleep(0.008)
          end
          var_value = rq_read_sta[index]

      elif (var_name == "FLT"):
          enter_critical
          rq_read_flt_req[index] = True
          exit_critical
          while(rq_read_flt_req[index]):
              sleep(0.008)
          end
          var_value = rq_read_flt[index]

      elif (var_name == "POS"):
          enter_critical
          rq_read_pos_req[index] = True
          exit_critical
          while(rq_read_pos_req[index]):
              sleep(0.008)
          end
          var_value = rq_read_pos[index]

      elif (var_name == "PRE"):
          enter_critical
          rq_read_pre_req[index] = True
          exit_critical
          while(rq_read_pre_req[index]):
              sleep(0.008)
          end
          var_value = rq_read_pre[index]

      elif (var_name == "LBP"):
          enter_critical
          rq_read_lbp_req[index] = True
          exit_critical
          while(rq_read_lbp_req[index]):
              sleep(0.008)
          end
          var_value = rq_read_lbp[index]

      elif (var_name == "LRD"):
          enter_critical
          rq_read_lrd_req[index] = True
          exit_critical
          while(rq_read_lrd_req[index]):
              sleep(0.008)
          end
          var_value = rq_read_lrd[index]

      elif (var_name == "LBL"):
          enter_critical
          rq_read_lbl_req[index] = True
          exit_critical
          while(rq_read_lbl_req[index]):
              sleep(0.008)
          end
          var_value = rq_read_lbl[index]

      elif (var_name == "LGN"):
          enter_critical
          rq_read_lgn_req[index] = True
          exit_critical
          while(rq_read_lgn_req[index]):
              sleep(0.008)
          end
          var_value = rq_read_lgn[index]

      elif (var_name == "MSC"):
          enter_critical
          rq_read_msc_req[index] = True
          exit_critical
          while(rq_read_msc_req[index]):
              sleep(0.008)
          end
          var_value = rq_read_msc[index]

      elif (var_name == "MOD"):
          enter_critical
          rq_read_mod_req[index] = True
          exit_critical
          while(rq_read_mod_req[index]):
              sleep(0.008)
          end
          var_value = rq_read_mod[index]

      elif (var_name == "NCY"):
          enter_critical
          rq_read_ncy_req[index] = True
          exit_critical
          while(rq_read_ncy_req[index]):
              sleep(0.008)
          end
          var_value = rq_read_ncy[index]

      elif (var_name == "PCO"):
          enter_critical
          rq_read_pco_req[index] = True
          exit_critical
          while(rq_read_pco_req[index]):
              sleep(0.008)
          end
          var_value = rq_read_pco[index]

      elif (var_name == "DST"):
          enter_critical
          rq_read_dst_req[index] = True
          exit_critical
          while(rq_read_dst_req[index]):
              sleep(0.008)
          end
          var_value = rq_read_dst[index]

      end

      return var_value
  end

  def rq_get_var_string(var_name, nbr_bytes, gripper_socket="1"):
      index = rq_socket_to_index(gripper_socket)
      var_value = ""

      enter_critical

      if (var_name == "SNU"):
          if(gripper_socket == "1"):
              var_value = rq_read_snu_1
          elif(gripper_socket == "2"):
              var_value = rq_read_snu_2
          elif(gripper_socket == "3"):
              var_value = rq_read_snu_3
          elif(gripper_socket == "4"):
              var_value = rq_read_snu_4
          end
      elif (var_name == "FWV"):
          if(gripper_socket == "1"):
              var_value = rq_read_fwv_1
          elif(gripper_socket == "2"):
              var_value = rq_read_fwv_2
          elif(gripper_socket == "3"):
              var_value = rq_read_fwv_3
          elif(gripper_socket == "4"):
              var_value = rq_read_fwv_4
          end
      elif (var_name == "VER"):
          if(gripper_socket == "1"):
              var_value = rq_read_ver_1
          elif(gripper_socket == "2"):
              var_value = rq_read_ver_2
          elif(gripper_socket == "3"):
              var_value = rq_read_ver_3
          elif(gripper_socket == "4"):
              var_value = rq_read_ver_4
          end
      end

      exit_critical

      return var_value
  end

  def rq_is_object_validated(gripper_selected, gripper_socket="1"):
      if(gripper_selected):
          if(rq_is_object_detected(gripper_socket)):
              return True
          else:
              return False
          end
      else:
          return True
      end
  end

  ############################################
  # normalized functions (maps 0-100 to 0-255)
  ############################################
  def rq_set_force_norm(force_norm, gripper_socket="1"):
      force_gripper = norm_to_gripper(force_norm)
      rq_set_force(force_gripper, gripper_socket)
  end

  def rq_set_speed_norm(speed_norm, gripper_socket="1"):
      speed_gripper = norm_to_gripper(speed_norm)
      rq_set_speed(speed_gripper, gripper_socket)
  end

  def rq_move_norm(pos_norm, gripper_socket="1"):
      pos_gripper = norm_to_gripper(pos_norm)
      rq_move(pos_gripper, gripper_socket)
  end

  def rq_move_and_wait_norm(pos_norm, gripper_socket="1"):
      pos_gripper = norm_to_gripper(pos_norm)
      rq_move_and_wait(pos_gripper, gripper_socket)
  end

  def rq_set_pos_norm(pos_norm, gripper_socket="1"):
      pos_gripper = norm_to_gripper(pos_norm)
      rq_set_pos(pos_gripper, gripper_socket)
  end

  def rq_current_pos_norm(gripper_socket="1"):
      pos_gripper = rq_current_pos(gripper_socket)
      pos_norm = gripper_to_norm(pos_gripper)
      return pos_norm
  end

  def gripper_to_norm(value_gripper):
      value_norm = (value_gripper / 255) * 100
      return floor(value_norm)
  end

  def norm_to_gripper(value_norm):
      value_gripper = (value_norm / 100) * 255
      return ceil(value_gripper)
  end

  def rq_get_position():
      return rq_current_pos_norm()
  end

  def rq_gripper_led_on(gripper_socket="1"):
      rq_set_var("LBP",0, gripper_socket)
  end

  def rq_gripper_led_off(gripper_socket="1"):
      rq_set_var("LBP",1, gripper_socket)
      rq_set_var("LRD",0, gripper_socket)
      rq_set_var("LBL",0, gripper_socket)
      rq_set_var("LGN",0, gripper_socket)
  end

  def rq_gripper_led_force_red(gripper_socket="1"):
      rq_set_var("LBP",1, gripper_socket)
      rq_set_var("LRD",1, gripper_socket)
      rq_set_var("LBL",0, gripper_socket)
      rq_set_var("LGN",0, gripper_socket)
  end

  def rq_gripper_led_force_blue(gripper_socket="1"):
      rq_set_var("LBP",1, gripper_socket)
      rq_set_var("LRD",0, gripper_socket)
      rq_set_var("LBL",1, gripper_socket)
      rq_set_var("LGN",0, gripper_socket)
  end

  def rq_gripper_led_force_green(gripper_socket="1"):
      rq_set_var("LBP",1, gripper_socket)
      rq_set_var("LRD",0, gripper_socket)
      rq_set_var("LBL",0, gripper_socket)
      rq_set_var("LGN",1, gripper_socket)
  end

  def rq_gripper_led_force_purple(gripper_socket="1"):
      rq_set_var("LBP",1, gripper_socket)
      rq_set_var("LRD",1, gripper_socket)
      rq_set_var("LBL",1, gripper_socket)
      rq_set_var("LGN",0, gripper_socket)
  end

  ############################################
  # mm/inches functions
  ############################################
  gripper_closed_norm = [100, 100, 100, 100]
  gripper_open_norm = [0, 0, 0, 0]
  gripper_closed_mm = [0, 0, 0, 0]
  gripper_open_mm = [50, 50, 50, 50]

  def rq_current_pos_mm(gripper_socket=1):
      pos_gripper = rq_current_pos(gripper_socket)
      pos_mm = gripper_to_mm(pos_gripper, gripper_socket)
      return round_value_2_dec(pos_mm)
  end

  def rq_current_pos_inches(gripper_socket=1):
      pos_gripper = rq_current_pos(gripper_socket)
      pos_mm = gripper_to_mm(pos_gripper, gripper_socket)
      pos_in = pos_mm / 25.4
      return round_value_2_dec(pos_in)
  end

  def rq_move_mm(pos_mm, gripper_socket=1):
      pos_gripper = mm_to_gripper(pos_mm, gripper_socket)
      rq_move(pos_gripper, gripper_socket)
  end

  def rq_move_and_wait_mm(pos_mm, gripper_socket=1):
      pos_gripper = mm_to_gripper(pos_mm, gripper_socket)
      rq_move_and_wait(pos_gripper, gripper_socket)
  end

  def rq_move_inches(pos_in, gripper_socket=1):
      pos_mm = pos_in * 25.4
      rq_move_mm(pos_mm, gripper_socket)
  end

  def rq_move_and_wait_inches(pos_in, gripper_socket=1):
      pos_mm = pos_in * 25.4
      rq_move_and_wait_mm(pos_mm, gripper_socket)
  end

  def get_closed_norm(gripper_socket):
      return gripper_closed_norm[gripper_socket - 1]
  end

  def get_open_norm(gripper_socket):
      return gripper_open_norm[gripper_socket - 1]
  end

  def get_closed_mm(gripper_socket):
      return gripper_closed_mm[gripper_socket - 1]
  end

  def get_open_mm(gripper_socket):
      return gripper_open_mm[gripper_socket - 1]
  end

  def set_closed_norm(closed_norm, gripper_socket):
      gripper_closed_norm[gripper_socket - 1] = closed_norm
  end

  def set_open_norm(open_norm, gripper_socket):
      gripper_open_norm[gripper_socket - 1] = open_norm
  end

  def set_closed_mm(closed_mm, gripper_socket):
      gripper_closed_mm[gripper_socket - 1] = closed_mm
  end

  def set_open_mm(open_mm, gripper_socket):
      gripper_open_mm[gripper_socket - 1] = open_mm
  end

  def gripper_to_mm(value_gripper, gripper_socket):
      closed_norm = get_closed_norm(gripper_socket)
      open_norm = get_open_norm(gripper_socket)
      closed_mm = get_closed_mm(gripper_socket)
      open_mm = get_open_mm(gripper_socket)

      value_norm = (value_gripper / 255) * 100

      slope = (closed_mm - open_mm) / (closed_norm - open_norm)
      value_mm = slope * (value_norm - closed_norm) + closed_mm

      if (value_mm > open_mm):
          value_mm_limited = open_mm
      elif (value_mm < closed_mm):
          value_mm_limited = closed_mm
      else:
          value_mm_limited = value_mm
      end

      return value_mm_limited
  end

  def mm_to_gripper(value_mm, gripper_socket):
      closed_norm = get_closed_norm(gripper_socket)
      open_norm = get_open_norm(gripper_socket)
      closed_mm = get_closed_mm(gripper_socket)
      open_mm = get_open_mm(gripper_socket)

      slope = (closed_norm - open_norm) / (closed_mm - open_mm)
      value_norm = (value_mm - closed_mm) * slope + closed_norm

      value_gripper = value_norm * 255 / 100

      if (value_gripper > 255):
          value_gripper_limited = 255
      elif (value_gripper < 0):
          value_gripper_limited = 0
      else:
          value_gripper_limited = round_value(value_gripper)
      end

      return value_gripper_limited
  end

  def round_value(value):
      value_mod = value % 1

      if(value_mod < 0.5):
          return floor(value)
      else:
          return ceil(value)
      end
  end

  def round_value_2_dec(value):
      value_x_100 = value * 100
      value_x_100_rounded = round_value(value_x_100)
      return value_x_100_rounded / 100
  end

  def clear_socket_buffer(gripper_socket="1", read_timeout = 0.1):
      rq_comm_clear_socket_buffer_enabled[rq_socket_to_index(gripper_socket)] = True
  end

  def rq_gripper_id_to_ascii(gripper_id):
      if(gripper_id == "1"):
          return 57
      elif(gripper_id == "2"):
          return 50
      elif(gripper_id == "3"):
          return 51
      elif(gripper_id == "4"):
          return 52
      end
  end

  def scale(value, rawRange, scaledRange):
      def computeSlope(inputRange, outputRange):
          outputRangeDelta = outputRange[1] - outputRange[0]
          inputRangeDelta = inputRange[1] - inputRange[0]

          if (inputRangeDelta == 0):
              return 0
          else:
              return outputRangeDelta / inputRangeDelta
          end
      end

      def computeIntercept(slope, inputRange, outputRange):
          return outputRange[0] - (slope * inputRange[0])
      end

      def clipScaledValue(outputScaledValue, outputRange):
          if (outputRange[0] < outputRange[1]):
              return clipWhenLowerLimitIsLessThanHigher(outputScaledValue, outputRange)
          else:
              return clipWhenLowerLimitIsGreaterThanHigherLimit(outputScaledValue, outputRange)
          end
      end

      def clipWhenLowerLimitIsGreaterThanHigherLimit(outputScaledValue, outputRange):
          if (outputScaledValue < outputRange[1]):
              return outputRange[1]
          elif (outputScaledValue > outputRange[0]):
              return outputRange[0]
          else:
              return outputScaledValue
          end
      end

      def clipWhenLowerLimitIsLessThanHigher(outputScaledValue, outputRange):
          if (outputScaledValue < outputRange[0]):
              return outputRange[0]
          elif (outputScaledValue > outputRange[1]):
              return outputRange[1]
          else:
              return outputScaledValue
          end
      end

      slope = computeSlope(rawRange, scaledRange)
      intercept = computeIntercept(slope, rawRange, scaledRange)
      scaledValue = slope * value + intercept
      return clipScaledValue(scaledValue, scaledRange)
  end

  def limit(value, range):
      return scale(value, range, range)
  end


  rq_init_comm_if_connected(9, "1")
  rq_init_comm_if_connected(2, "2")
  rq_init_comm_if_connected(3, "3")
  rq_init_comm_if_connected(4, "4")
  rq_print_connected_grippers()
  rq_gripper_communication_thread = run rq_gripper_communication()
  set_closed_norm(90.19607843137254, 1)
  set_open_norm(1.1764705882352942, 1)
  set_closed_mm(0.0, 1)
  set_open_mm(86.0, 1)
  set_closed_norm(100.0, 2)
  set_open_norm(0.0, 2)
  set_closed_mm(0.0, 2)
  set_open_mm(50.0, 2)
  set_closed_norm(100.0, 3)
  set_open_norm(0.0, 3)
  set_closed_mm(0.0, 3)
  set_open_mm(50.0, 3)
  set_closed_norm(100.0, 4)
  set_open_norm(0.0, 4)
  set_closed_mm(0.0, 4)
  set_open_mm(50.0, 4)
  rq_current_limit_enabled = False
  while(not rq_gripper_communication_thread_started):
      sleep(0.008)
  end
  # end: URCap Installation Node
  $ 1 "BeforeStart"
  $ 2 "Script: Setup.script"
  #  This program is for setting up the robot vision system using
  #  Keyence's vision sensor.
  #  Please do not use it for purposes other than its original
  #  intended purpose.
  #  With regard to robot operation, please use the robot while
  #  following the precautions stated in the "User's Manual".
  #
  # Copyright (c) 2015 KEYENCE CORPORATION. All rights reserved.


  def CUR_SetUpCamera(CAM, IP_Address, Port):
  # Pass parameters to global variables.
    global Camera = CAM
    varmsg("Camera", Camera)

    global IP = IP_Address
    varmsg("IP", IP)

    global TelPort = Port
    varmsg("TelPort", TelPort)

    global Version = 3000000
    varmsg("Version", Version)

    global DiscID = 120
    varmsg("DiscID", DiscID)

    global Speed = 10
    varmsg("Speed", Speed)

    global Accel = 100
    varmsg("Accel", Accel)

    global MaxRealSpeed = 0.3
    global MaxRealAccel = 0.3

  end


  def CUR_InitComm(CAM):
  # Open the connection.
    global connected = False
    while (not  connected):
      global connected = socket_open(IP, TelPort, Camera)	# Establish connection to camera
      varmsg("connected", connected)						# server via Telnet
    end
    return connected
  end


  def CUR_ProcCommand(CAM):
  # Process a command.
    global Camera = CAM
    varmsg("Camera", Camera)
    global nComID = 0
    varmsg("nComID", nComID)
    global nOprtID = 0
    varmsg("nOprtID", nOprtID)
    global nReqID = 0
    varmsg("nReqID", nReqID)
    local nResRslt = 0
    varmsg("nResRslt", nResRslt)
    global Com = socket_read_ascii_float(13, Camera)
    varmsg("Com", Com)
    local P0 = 0
    local P1 = 0
    local P2 = 0
    local P3 = 0
    local P4 = 0
    local P5 = 0
    local P6 = 0
    local P7 = 0
    local P8 = 0

    local argNum = floor(Com[0])

    if argNum >= 1:
      nComID = floor(Com[1])
    end
    if argNum >= 2:
      nOprtID = floor(Com[2])
    end
    if argNum >= 3:
      nReqID = floor(Com[3])
    end
    if argNum >= 4:
      P0 = floor(Com[4])
    end
    if argNum >= 5:
      P1 = floor(Com[5])
    end
    if argNum >= 6:
      P2 = floor(Com[6])
    end
    if argNum >= 7:
      P3 = floor(Com[7])
    end
    if argNum >= 8:
      P4 = floor(Com[8])
    end
    if argNum >= 9:
      P5 = floor(Com[9])
    end
    if argNum >= 10:
      P6 = floor(Com[10])
    end
    if argNum >= 11:
      P7 = floor(Com[11])
    end
    if argNum >= 12:
      P8 = floor(Com[12])
    end

    if argNum == 0:
  # Read failed or timeout
      return 0
    elif nComID != 3:
  # Invalid command number
      OutputError(nOprtID, nReqID, nResRslt)
      return 1
    end

    if nOprtID == 1:
  # Echo reply
      Sum = P2
      nResRslt = ProcEcho(nOprtID, nReqID, Sum, P0, P1)

    elif nOprtID == 2:
  # Get Parameters
      Sum = P0
      nResRslt = ProcGetParam(nOprtID, nReqID, Sum)

    elif nOprtID == 3:
  # Set Parameters
      Sum = P5
      nResRslt = ProcSetParam(nOprtID, nReqID, Sum, P0, P1, P2, P3, P4)

    elif nOprtID == 4:
  # Get current position
      Sum = P0
      nResRslt = ProcGetPos(nOprtID, nReqID, Sum)

    elif nOprtID == 5:
  # Move relatively
      Sum = P8
      nResRslt = ProcMoveRel(nOprtID, nReqID, Sum, P0, P1, P2, P3, P4, P5, P6, P7)

    elif nOprtID == 6:
  # Move absolutely
      Sum = P6
      nResRslt = ProcMoveAbs(nOprtID, nReqID, Sum, P0, P1, P2, P3, P4, P5)

    elif nOprtID == 7:
  # Get version
      Sum = P0
      nResRslt = ProcGetVer(nOprtID, nReqID, Sum)

    elif nOprtID == 8:
  # Get tool coordinate
      Sum = P1
      nResRslt = ProcGetTool(nOprtID, nReqID, Sum, P0)

    elif nOprtID == 9:
  # Get current position (high-precision)
      Sum = P0
      nResRslt = ProcGetPosHp(nOprtID, nReqID, Sum)

    elif nOprtID == 10:
  # Move relatively (high-precision)
      Sum = P8
      nResRslt = ProcMoveRelHp(nOprtID, nReqID, Sum, P0, P1, P2, P3, P4, P5, P6, P7)

    elif nOprtID == 11:
  # Move absolutely (high-precision)
      Sum = P6
      nResRslt = ProcMoveAbsHp(nOprtID, nReqID, Sum, P0, P1, P2, P3, P4, P5)

    elif nOprtID == 12:
  # Get current joint position
      Sum = P0
      nResRslt = ProcGetJPos(nOprtID, nReqID, Sum)

    elif nOprtID == 13:
  # Get user coordinate
      Sum = P0
      nResRslt = ProcGetUser(nOprtID, nReqID, Sum)

    elif nOprtID == 14:
  # Move relatively (joint)
      Sum = P6
      nResRslt = ProcMoveJRel(nOprtID, nReqID, Sum, P0, P1, P2, P3, P4, P5)

    elif nOprtID == 15:
  # Move absolutely (joint)
      Sum = P6
      nResRslt = ProcMoveJAbs(nOprtID, nReqID, Sum, P0, P1, P2, P3, P4, P5)

    else:
      nResRslt = 1

    end

    if nResRslt != 0:
      OutputError(nOprtID, nReqID, nResRslt)
    end

    return nResRslt
  end


  def CUR_CloseComm(CAM):
  # Close the connection.
    global Camera = CAM
    varmsg("Camera", Camera)
    socket_close(Camera)
  end


  # Echo reply
  def ProcEcho(nOprtID, nReqID, Sum, P0, P1):
  # Result
    local nParamSum = nOprtID + nReqID + P0 + P1
    local nResRslt = 0
    if Sum != nParamSum:
      nResRslt = 1
      return nResRslt
    end
  # Process
    local O0 = P0
    local O1 = P1
  # Conversion
    local nResSum = O0 + O1
    nResSum = nResSum + nOprtID + nReqID + nResRslt

    socket_send_string("CRBT,", Camera)
    socket_send_string(nOprtID, Camera)
    socket_send_string(",", Camera)
    socket_send_string(nReqID, Camera)
    socket_send_string(",", Camera)
    socket_send_string(nResRslt, Camera)
    socket_send_string(",", Camera)
    socket_send_string(O0, Camera)
    socket_send_string(",", Camera)
    socket_send_string(O1, Camera)
    socket_send_string(",", Camera)
    socket_send_string(nResSum, Camera)
    socket_send_crlf(Camera)

    return nResRslt
  end


  # Get parameters
  def ProcGetParam(nOprtID, nReqID, Sum):
  # Result
    local nParamSum = nOprtID + nReqID
    local nResRslt = 0
    if Sum != nParamSum:
      nResRslt = 1
      return nResRslt
    end
  # Process
    local O0 = 0
    local O1 = 0
    local O2 = 0
    local O3 = Speed
    local O4 = Accel
  # Conversion
    nResSum = O0 + O1 + O2 + O3 + O4
    nResSum = nResSum + nOprtID + nReqID + nResRslt

    socket_send_string("CRBT,", Camera)
    socket_send_string(nOprtID, Camera)
    socket_send_string(",", Camera)
    socket_send_string(nReqID, Camera)
    socket_send_string(",", Camera)
    socket_send_string(nResRslt, Camera)
    socket_send_string(",", Camera)
    socket_send_string(O0, Camera)
    socket_send_string(",", Camera)
    socket_send_string(O1, Camera)
    socket_send_string(",", Camera)
    socket_send_string(O2, Camera)
    socket_send_string(",", Camera)
    socket_send_string(O3, Camera)
    socket_send_string(",", Camera)
    socket_send_string(O4, Camera)
    socket_send_string(",", Camera)
    socket_send_string(nResSum, Camera)
    socket_send_crlf(Camera)

    return nResRslt
  end



  # Set parameters
  def ProcSetParam(nOprtID, nReqID, Sum, P0, P1, P2, P3, P4):
  # Result
    local nParamSum = nOprtID + nReqID + P0 + P1 + P2 + P3 + P4
    local nResRslt = 0
    if Sum != nParamSum:
      nResRslt = 1
      return nResRslt
    end
  # Process
    if P1 != 0:
      nResRslt = 2
    end
    if P2 != 0:
      nResRslt = 2
    end
    Speed = P3
    Accel = P4

    local O0 = 0
    local O1 = 0
    local O2 = 0
    local O3 = Speed
    local O4 = Accel
  # Conversion
    local nResSum = O0 + O1 + O2 + O3 + O4
    nResSum = nResSum + nOprtID + nReqID + nResRslt

    socket_send_string("CRBT,", Camera)
    socket_send_string(nOprtID, Camera)
    socket_send_string(",", Camera)
    socket_send_string(nReqID, Camera)
    socket_send_string(",", Camera)
    socket_send_string(nResRslt, Camera)
    socket_send_string(",", Camera)
    socket_send_string(O0, Camera)
    socket_send_string(",", Camera)
    socket_send_string(O1, Camera)
    socket_send_string(",", Camera)
    socket_send_string(O2, Camera)
    socket_send_string(",", Camera)
    socket_send_string(O3, Camera)
    socket_send_string(",", Camera)
    socket_send_string(O4, Camera)
    socket_send_string(",", Camera)
    socket_send_string(nResSum, Camera)
    socket_send_crlf(Camera)

    return nResRslt
  end



  # Get current position
  def ProcGetPos(nOprtID, nReqID, Sum):
  # Result
    local nParamSum = nOprtID + nReqID
    local nResRslt = 0
    if Sum != nParamSum:
      nResRslt = 1
      return nResRslt
    end
  # Process
    local CurrentPos = get_actual_tcp_pose_RPY()
    local O0 = floor(CurrentPos[0] * 1000000.0 + 0.5)
    local O1 = floor(CurrentPos[1] * 1000000.0 + 0.5)
    local O2 = floor(CurrentPos[2] * 1000000.0 + 0.5)
    local O3 = floor(Key_r2d(CurrentPos[3]) * 10.0 + 0.5)
    local O4 = floor(Key_r2d(CurrentPos[4]) * 10.0 + 0.5)
    local O5 = floor(Key_r2d(CurrentPos[5]) * 10.0 + 0.5)
  # Conversion
    local nResSum = O0 + O1 + O2 + O3 + O4 + O5
    nResSum = nResSum + nOprtID + nReqID + nResRslt

    socket_send_string("CRBT,", Camera)
    socket_send_string(nOprtID, Camera)
    socket_send_string(",", Camera)
    socket_send_string(nReqID, Camera)
    socket_send_string(",", Camera)
    socket_send_string(nResRslt, Camera)
    socket_send_string(",", Camera)
    socket_send_string(O0, Camera)
    socket_send_string(",", Camera)
    socket_send_string(O1, Camera)
    socket_send_string(",", Camera)
    socket_send_string(O2, Camera)
    socket_send_string(",", Camera)
    socket_send_string(O3, Camera)
    socket_send_string(",", Camera)
    socket_send_string(O4, Camera)
    socket_send_string(",", Camera)
    socket_send_string(O5, Camera)
    socket_send_string(",", Camera)
    socket_send_string(nResSum, Camera)
    socket_send_crlf(Camera)

    return nResRslt
  end



  # Move relatively
  def ProcMoveRel(nOprtID, nReqID, Sum, P0, P1, P2, P3, P4, P5, P6, P7):
  # Result
    local nParamSum = nOprtID + nReqID + P0 + P1 + P2 + P3 + P4 + P5 + P6 + P7
    local nResRslt = 0
    if Sum != nParamSum:
      nResRslt = 1
      return nResRslt
    end
  # Process
    local CurrentPos = get_actual_tcp_pose_RPY()
    A0 = P0 / 1000000.0
    A1 = P1 / 1000000.0
    A2 = P2 / 1000000.0
    A3 = d2r(P3) / 10.0
    A4 = d2r(P4) / 10.0
    A5 = d2r(P5) / 10.0
    local Vec = p[A0, A1, A2, A3, A4, A5]
    local Pos = pose_add_RPY(CurrentPos, Vec)
    MoveRPY(Pos)

    CurrentPos = get_actual_tcp_pose_RPY()
    local O0 = floor(CurrentPos[0] * 1000000.0 + 0.5)
    local O1 = floor(CurrentPos[1] * 1000000.0 + 0.5)
    local O2 = floor(CurrentPos[2] * 1000000.0 + 0.5)
    local O3 = floor(Key_r2d(CurrentPos[3]) * 10.0 + 0.5)
    local O4 = floor(Key_r2d(CurrentPos[4]) * 10.0 + 0.5)
    local O5 = floor(Key_r2d(CurrentPos[5]) * 10.0 + 0.5)
  # Conversion
    local nResSum = O0 + O1 + O2 + O3 + O4 + O5
    nResSum = nResSum + nOprtID + nReqID + nResRslt

    socket_send_string("CRBT,", Camera)
    socket_send_string(nOprtID, Camera)
    socket_send_string(",", Camera)
    socket_send_string(nReqID, Camera)
    socket_send_string(",", Camera)
    socket_send_string(nResRslt, Camera)
    socket_send_string(",", Camera)
    socket_send_string(O0, Camera)
    socket_send_string(",", Camera)
    socket_send_string(O1, Camera)
    socket_send_string(",", Camera)
    socket_send_string(O2, Camera)
    socket_send_string(",", Camera)
    socket_send_string(O3, Camera)
    socket_send_string(",", Camera)
    socket_send_string(O4, Camera)
    socket_send_string(",", Camera)
    socket_send_string(O5, Camera)
    socket_send_string(",", Camera)
    socket_send_string(nResSum, Camera)
    socket_send_crlf(Camera)

    return nResRslt
  end



  # Move absolutely
  def ProcMoveAbs(nOprtID, nReqID, Sum, P0, P1, P2, P3, P4, P5):
  # Result
    local nParamSum = nOprtID + nReqID + P0 + P1 + P2 + P3 + P4 + P5
    local nResRslt = 0
    if Sum != nParamSum:
      nResRslt = 1
      return nResRslt
    end
  # Process
    A0 = P0 / 1000000.0
    A1 = P1 / 1000000.0
    A2 = P2 / 1000000.0
    A3 = d2r(P3) / 10.0
    A4 = d2r(P4) / 10.0
    A5 = d2r(P5) / 10.0
    local Pos = p[A0, A1, A2, A3, A4, A5]
    MoveRPY(Pos)

    local CurrentPos = get_actual_tcp_pose_RPY()
    local O0 = floor(CurrentPos[0] * 1000000.0 + 0.5)
    local O1 = floor(CurrentPos[1] * 1000000.0 + 0.5)
    local O2 = floor(CurrentPos[2] * 1000000.0 + 0.5)
    local O3 = floor(Key_r2d(CurrentPos[3]) * 10.0 + 0.5)
    local O4 = floor(Key_r2d(CurrentPos[4]) * 10.0 + 0.5)
    local O5 = floor(Key_r2d(CurrentPos[5]) * 10.0 + 0.5)
  # Conversion
    local nResSum = O0 + O1 + O2 + O3 + O4 + O5
    nResSum = nResSum + nOprtID + nReqID + nResRslt

    socket_send_string("CRBT,", Camera)
    socket_send_string(nOprtID, Camera)
    socket_send_string(",", Camera)
    socket_send_string(nReqID, Camera)
    socket_send_string(",", Camera)
    socket_send_string(nResRslt, Camera)
    socket_send_string(",", Camera)
    socket_send_string(O0, Camera)
    socket_send_string(",", Camera)
    socket_send_string(O1, Camera)
    socket_send_string(",", Camera)
    socket_send_string(O2, Camera)
    socket_send_string(",", Camera)
    socket_send_string(O3, Camera)
    socket_send_string(",", Camera)
    socket_send_string(O4, Camera)
    socket_send_string(",", Camera)
    socket_send_string(O5, Camera)
    socket_send_string(",", Camera)
    socket_send_string(nResSum, Camera)
    socket_send_crlf(Camera)

    return nResRslt
  end


  # Get version
  def ProcGetVer(nOprtID, nReqID, Sum):
  # Result
    local nParamSum = nOprtID + nReqID
    local nResRslt = 0
    if Sum != nParamSum:
      nResRslt = 1
      return nResRslt
    end
  # Process
    local O0 = Version
    local O1 = DiscID
  # Conversion
    nResSum = O0 + O1
    nResSum = nResSum + nOprtID + nReqID + nResRslt

    socket_send_string("CRBT,", Camera)
    socket_send_string(nOprtID, Camera)
    socket_send_string(",", Camera)
    socket_send_string(nReqID, Camera)
    socket_send_string(",", Camera)
    socket_send_string(nResRslt, Camera)
    socket_send_string(",", Camera)
    socket_send_string(O0, Camera)
    socket_send_string(",", Camera)
    socket_send_string(O1, Camera)
    socket_send_string(",", Camera)
    socket_send_string(nResSum, Camera)
    socket_send_crlf(Camera)

    return nResRslt
  end



  # Get tool coordinate (not supported)
  def ProcGetTool(nOprtID, nReqID, Sum, P0):
  # Result
    local nParamSum = nOprtID + nReqID
    local nResRslt = 0
    if Sum != nParamSum:
      nResRslt = 1
      return nResRslt
    end
  # Process
    nResRslt = 3
    local O0 = 0
    local O1 = 0
    local O2 = 0
    local O3 = 0
    local O4 = 0
    local O5 = 0
  # Conversion
    local nResSum = O0 + O1 + O2 + O3 + O4 + O5
    nResSum = nResSum + nOprtID + nReqID + nResRslt

    socket_send_string("CRBT,", Camera)
    socket_send_string(nOprtID, Camera)
    socket_send_string(",", Camera)
    socket_send_string(nReqID, Camera)
    socket_send_string(",", Camera)
    socket_send_string(nResRslt, Camera)
    socket_send_string(",", Camera)
    socket_send_string(O0, Camera)
    socket_send_string(",", Camera)
    socket_send_string(O1, Camera)
    socket_send_string(",", Camera)
    socket_send_string(O2, Camera)
    socket_send_string(",", Camera)
    socket_send_string(O3, Camera)
    socket_send_string(",", Camera)
    socket_send_string(O4, Camera)
    socket_send_string(",", Camera)
    socket_send_string(O5, Camera)
    socket_send_string(",", Camera)
    socket_send_string(nResSum, Camera)
    socket_send_crlf(Camera)

    return nResRslt
  end



  # Get user coordinate (not supported)
  def ProcGetUser(nOprtID, nReqID, Sum):
  # Result
    local nParamSum = nOprtID + nReqID
    local nResRslt = 0
    if Sum != nParamSum:
      nResRslt = 1
      return nResRslt
    end
  # Process
    nResRslt = 2
    local O0 = 0
    local O1 = 0
    local O2 = 0
    local O3 = 0
    local O4 = 0
    local O5 = 0
  # Conversion
    local nResSum = O0 + O1 + O2 + O3 + O4 + O5
    nResSum = nResSum + nOprtID + nReqID + nResRslt

    socket_send_string("CRBT,", Camera)
    socket_send_string(nOprtID, Camera)
    socket_send_string(",", Camera)
    socket_send_string(nReqID, Camera)
    socket_send_string(",", Camera)
    socket_send_string(nResRslt, Camera)
    socket_send_string(",", Camera)
    socket_send_string(O0, Camera)
    socket_send_string(",", Camera)
    socket_send_string(O1, Camera)
    socket_send_string(",", Camera)
    socket_send_string(O2, Camera)
    socket_send_string(",", Camera)
    socket_send_string(O3, Camera)
    socket_send_string(",", Camera)
    socket_send_string(O4, Camera)
    socket_send_string(",", Camera)
    socket_send_string(O5, Camera)
    socket_send_string(",", Camera)
    socket_send_string(nResSum, Camera)
    socket_send_crlf(Camera)

    return nResRslt
  end


  # Get current position (high-precision)
  def ProcGetPosHp(nOprtID, nReqID, Sum):
  # Result
    local nParamSum = nOprtID + nReqID
    local nResRslt = 0
    if Sum != nParamSum:
      nResRslt = 1
      return nResRslt
    end
  # Process
    local CurrentPos = get_actual_tcp_pose_RPY()
    local O0 = floor(CurrentPos[0] * 1000000.0 + 0.5)
    local O1 = floor(CurrentPos[1] * 1000000.0 + 0.5)
    local O2 = floor(CurrentPos[2] * 1000000.0 + 0.5)
    local O3 = floor(Key_r2d(CurrentPos[3]) * 1000.0 + 0.5)
    local O4 = floor(Key_r2d(CurrentPos[4]) * 1000.0 + 0.5)
    local O5 = floor(Key_r2d(CurrentPos[5]) * 1000.0 + 0.5)
  # Conversion
    local nResSum = O0 + O1 + O2 + O3 + O4 + O5
    nResSum = nResSum + nOprtID + nReqID + nResRslt

    socket_send_string("CRBT,", Camera)
    socket_send_string(nOprtID, Camera)
    socket_send_string(",", Camera)
    socket_send_string(nReqID, Camera)
    socket_send_string(",", Camera)
    socket_send_string(nResRslt, Camera)
    socket_send_string(",", Camera)
    socket_send_string(O0, Camera)
    socket_send_string(",", Camera)
    socket_send_string(O1, Camera)
    socket_send_string(",", Camera)
    socket_send_string(O2, Camera)
    socket_send_string(",", Camera)
    socket_send_string(O3, Camera)
    socket_send_string(",", Camera)
    socket_send_string(O4, Camera)
    socket_send_string(",", Camera)
    socket_send_string(O5, Camera)
    socket_send_string(",", Camera)
    socket_send_string(nResSum, Camera)
    socket_send_crlf(Camera)

    return nResRslt
  end



  # Get current joint position
  def ProcGetJPos(nOprtID, nReqID, Sum):
  # Result
    local nParamSum = nOprtID + nReqID
    local nResRslt = 0
    if Sum != nParamSum:
      nResRslt = 1
      return nResRslt
    end
  # Process
    local CurrentPos = get_actual_joint_positions()
    local O0 = floor(r2d(CurrentPos[0]) * 1000.0 + 0.5)
    local O1 = floor(r2d(CurrentPos[1]) * 1000.0 + 0.5)
    local O2 = floor(r2d(CurrentPos[2]) * 1000.0 + 0.5)
    local O3 = floor(r2d(CurrentPos[3]) * 1000.0 + 0.5)
    local O4 = floor(r2d(CurrentPos[4]) * 1000.0 + 0.5)
    local O5 = floor(r2d(CurrentPos[5]) * 1000.0 + 0.5)
  # Conversion
    local nResSum = O0 + O1 + O2 + O3 + O4 + O5
    nResSum = nResSum + nOprtID + nReqID + nResRslt

    socket_send_string("CRBT,", Camera)
    socket_send_string(nOprtID, Camera)
    socket_send_string(",", Camera)
    socket_send_string(nReqID, Camera)
    socket_send_string(",", Camera)
    socket_send_string(nResRslt, Camera)
    socket_send_string(",", Camera)
    socket_send_string(O0, Camera)
    socket_send_string(",", Camera)
    socket_send_string(O1, Camera)
    socket_send_string(",", Camera)
    socket_send_string(O2, Camera)
    socket_send_string(",", Camera)
    socket_send_string(O3, Camera)
    socket_send_string(",", Camera)
    socket_send_string(O4, Camera)
    socket_send_string(",", Camera)
    socket_send_string(O5, Camera)
    socket_send_string(",", Camera)
    socket_send_string(nResSum, Camera)
    socket_send_crlf(Camera)

    return nResRslt
  end



  # Move relatively (high-precision)
  def ProcMoveRelHp(nOprtID, nReqID, Sum, P0, P1, P2, P3, P4, P5, P6, P7):
  # Result
    local nParamSum = nOprtID + nReqID + P0 + P1 + P2 + P3 + P4 + P5 + P6 + P7
    local nResRslt = 0
    if Sum != nParamSum:
      nResRslt = 1
      return nResRslt
    end
  # Process
    local CurrentPos = get_actual_tcp_pose_RPY()
    A0 = P0 / 1000000.0
    A1 = P1 / 1000000.0
    A2 = P2 / 1000000.0
    A3 = d2r(P3) / 1000.0
    A4 = d2r(P4) / 1000.0
    A5 = d2r(P5) / 1000.0
    local Vec = p[A0, A1, A2, A3, A4, A5]
    local Pos = pose_add_RPY(CurrentPos, Vec)
    MoveRPY(Pos)

    CurrentPos = get_actual_tcp_pose_RPY()
    local O0 = floor(CurrentPos[0] * 1000000.0 + 0.5)
    local O1 = floor(CurrentPos[1] * 1000000.0 + 0.5)
    local O2 = floor(CurrentPos[2] * 1000000.0 + 0.5)
    local O3 = floor(Key_r2d(CurrentPos[3]) * 1000.0 + 0.5)
    local O4 = floor(Key_r2d(CurrentPos[4]) * 1000.0 + 0.5)
    local O5 = floor(Key_r2d(CurrentPos[5]) * 1000.0 + 0.5)
  # Conversion
    local nResSum = O0 + O1 + O2 + O3 + O4 + O5
    nResSum = nResSum + nOprtID + nReqID + nResRslt

    socket_send_string("CRBT,", Camera)
    socket_send_string(nOprtID, Camera)
    socket_send_string(",", Camera)
    socket_send_string(nReqID, Camera)
    socket_send_string(",", Camera)
    socket_send_string(nResRslt, Camera)
    socket_send_string(",", Camera)
    socket_send_string(O0, Camera)
    socket_send_string(",", Camera)
    socket_send_string(O1, Camera)
    socket_send_string(",", Camera)
    socket_send_string(O2, Camera)
    socket_send_string(",", Camera)
    socket_send_string(O3, Camera)
    socket_send_string(",", Camera)
    socket_send_string(O4, Camera)
    socket_send_string(",", Camera)
    socket_send_string(O5, Camera)
    socket_send_string(",", Camera)
    socket_send_string(nResSum, Camera)
    socket_send_crlf(Camera)

    return nResRslt
  end



  # Move relatively (joint)
  def ProcMoveJRel(nOprtID, nReqID, Sum, P0, P1, P2, P3, P4, P5):
  # Result
    local nParamSum = nOprtID + nReqID + P0 + P1 + P2 + P3 + P4 + P5
    local nResRslt = 0
    if Sum != nParamSum:
      nResRslt = 1
      return nResRslt
    end
  # Process
    local CurrentPos = get_actual_joint_positions()
    A0 = d2r(P0 / 1000.0)
    A1 = d2r(P1 / 1000.0)
    A2 = d2r(P2 / 1000.0)
    A3 = d2r(P3 / 1000.0)
    A4 = d2r(P4 / 1000.0)
    A5 = d2r(P5 / 1000.0)
    local Vec = p[A0, A1, A2, A3, A4, A5]
    local Pos = pose_add_RPY(CurrentPos, Vec)
    MoveJ_(Pos)

    CurrentPos = get_actual_joint_positions()
    local O0 = floor(r2d(CurrentPos[0]) * 1000.0 + 0.5)
    local O1 = floor(r2d(CurrentPos[1]) * 1000.0 + 0.5)
    local O2 = floor(r2d(CurrentPos[2]) * 1000.0 + 0.5)
    local O3 = floor(r2d(CurrentPos[3]) * 1000.0 + 0.5)
    local O4 = floor(r2d(CurrentPos[4]) * 1000.0 + 0.5)
    local O5 = floor(r2d(CurrentPos[5]) * 1000.0 + 0.5)
  # Conversion
    local nResSum = O0 + O1 + O2 + O3 + O4 + O5
    nResSum = nResSum + nOprtID + nReqID + nResRslt

    socket_send_string("CRBT,", Camera)
    socket_send_string(nOprtID, Camera)
    socket_send_string(",", Camera)
    socket_send_string(nReqID, Camera)
    socket_send_string(",", Camera)
    socket_send_string(nResRslt, Camera)
    socket_send_string(",", Camera)
    socket_send_string(O0, Camera)
    socket_send_string(",", Camera)
    socket_send_string(O1, Camera)
    socket_send_string(",", Camera)
    socket_send_string(O2, Camera)
    socket_send_string(",", Camera)
    socket_send_string(O3, Camera)
    socket_send_string(",", Camera)
    socket_send_string(O4, Camera)
    socket_send_string(",", Camera)
    socket_send_string(O5, Camera)
    socket_send_string(",", Camera)
    socket_send_string(nResSum, Camera)
    socket_send_crlf(Camera)

    return nResRslt
  end



  # Move absolutely (joint)
  def ProcMoveJAbs(nOprtID, nReqID, Sum, P0, P1, P2, P3, P4, P5):
  # Result
    local nParamSum = nOprtID + nReqID + P0 + P1 + P2 + P3 + P4 + P5
    local nResRslt = 0
    if Sum != nParamSum:
      nResRslt = 1
      return nResRslt
    end
  # Process
    A0 = d2r(P0 / 1000.0)
    A1 = d2r(P1 / 1000.0)
    A2 = d2r(P2 / 1000.0)
    A3 = d2r(P3 / 1000.0)
    A4 = d2r(P4 / 1000.0)
    A5 = d2r(P5 / 1000.0)
    local Pos = p[A0, A1, A2, A3, A4, A5]
    MoveJ_(Pos)

    local CurrentPos = get_actual_joint_positions()
    local O0 = floor(r2d(CurrentPos[0]) * 1000.0 + 0.5)
    local O1 = floor(r2d(CurrentPos[1]) * 1000.0 + 0.5)
    local O2 = floor(r2d(CurrentPos[2]) * 1000.0 + 0.5)
    local O3 = floor(r2d(CurrentPos[3]) * 1000.0 + 0.5)
    local O4 = floor(r2d(CurrentPos[4]) * 1000.0 + 0.5)
    local O5 = floor(r2d(CurrentPos[5]) * 1000.0 + 0.5)
  # Conversion
    local nResSum = O0 + O1 + O2 + O3 + O4 + O5
    nResSum = nResSum + nOprtID + nReqID + nResRslt

    socket_send_string("CRBT,", Camera)
    socket_send_string(nOprtID, Camera)
    socket_send_string(",", Camera)
    socket_send_string(nReqID, Camera)
    socket_send_string(",", Camera)
    socket_send_string(nResRslt, Camera)
    socket_send_string(",", Camera)
    socket_send_string(O0, Camera)
    socket_send_string(",", Camera)
    socket_send_string(O1, Camera)
    socket_send_string(",", Camera)
    socket_send_string(O2, Camera)
    socket_send_string(",", Camera)
    socket_send_string(O3, Camera)
    socket_send_string(",", Camera)
    socket_send_string(O4, Camera)
    socket_send_string(",", Camera)
    socket_send_string(O5, Camera)
    socket_send_string(",", Camera)
    socket_send_string(nResSum, Camera)
    socket_send_crlf(Camera)

    return nResRslt
  end



  # Move absolutely (high-precision)
  def ProcMoveAbsHp(nOprtID, nReqID, Sum, P0, P1, P2, P3, P4, P5):
  # Result
    local nParamSum = nOprtID + nReqID + P0 + P1 + P2 + P3 + P4 + P5
    local nResRslt = 0
    if Sum != nParamSum:
      nResRslt = 1
      return nResRslt
    end
  # Process
    A0 = P0 / 1000000.0
    A1 = P1 / 1000000.0
    A2 = P2 / 1000000.0
    A3 = d2r(P3) / 1000.0
    A4 = d2r(P4) / 1000.0
    A5 = d2r(P5) / 1000.0
    local Pos = p[A0, A1, A2, A3, A4, A5]
    MoveRPY(Pos)

    local CurrentPos = get_actual_tcp_pose_RPY()
    local O0 = floor(CurrentPos[0] * 1000000.0 + 0.5)
    local O1 = floor(CurrentPos[1] * 1000000.0 + 0.5)
    local O2 = floor(CurrentPos[2] * 1000000.0 + 0.5)
    local O3 = floor(Key_r2d(CurrentPos[3]) * 1000.0 + 0.5)
    local O4 = floor(Key_r2d(CurrentPos[4]) * 1000.0 + 0.5)
    local O5 = floor(Key_r2d(CurrentPos[5]) * 1000.0 + 0.5)
  # Conversion
    local nResSum = O0 + O1 + O2 + O3 + O4 + O5
    nResSum = nResSum + nOprtID + nReqID + nResRslt

    socket_send_string("CRBT,", Camera)
    socket_send_string(nOprtID, Camera)
    socket_send_string(",", Camera)
    socket_send_string(nReqID, Camera)
    socket_send_string(",", Camera)
    socket_send_string(nResRslt, Camera)
    socket_send_string(",", Camera)
    socket_send_string(O0, Camera)
    socket_send_string(",", Camera)
    socket_send_string(O1, Camera)
    socket_send_string(",", Camera)
    socket_send_string(O2, Camera)
    socket_send_string(",", Camera)
    socket_send_string(O3, Camera)
    socket_send_string(",", Camera)
    socket_send_string(O4, Camera)
    socket_send_string(",", Camera)
    socket_send_string(O5, Camera)
    socket_send_string(",", Camera)
    socket_send_string(nResSum, Camera)
    socket_send_crlf(Camera)

    return nResRslt
  end



  # Output an error message
  def OutputError(nOprtID, nReqID, nResRslt):
  # Conversion
    nResSum = nOprtID + nReqID + nResRslt

    socket_send_string("CRBT,", Camera)
    socket_send_string(nOprtID, Camera)
    socket_send_string(",", Camera)
    socket_send_string(nReqID, Camera)
    socket_send_string(",", Camera)
    socket_send_string(nResRslt, Camera)
    socket_send_string(",", Camera)
    socket_send_string(nResSum, Camera)
    socket_send_crlf(Camera)

    return nResRslt
  end


  # Send CRLF
  def socket_send_crlf(CAM):
    global Camera = CAM

    socket_send_byte(13, Camera)				# Carriage Return 0Dhex 13dec
    socket_send_byte(10, Camera)				# Line Feed 0Ahex 10dec
  end


  # Conversion (Radian to Degree)
  def Key_r2d(value):
    local r2d_ratio = 57.29577951
    return r2d_ratio * value
  end

  # Move
  def MoveRPY(Pos):
    local RealAccel = Accel * MaxRealAccel / 100.0
    local RealSpeed = Speed * MaxRealSpeed / 100.0

    A = RPY_to_AxisAngle(Pos)
    movel(A, RealAccel, RealSpeed)
  end

  # MoveJ
  def MoveJ_(Pos):
    local RealAccel = Accel * MaxRealAccel / 100.0
    local RealSpeed = Speed * MaxRealSpeed / 100.0

    movej(Pos, RealAccel, RealSpeed)
  end

  # Conversion (RPY to AxisAngle)
  def RPY_to_AxisAngle(R):
    Rx = R[3] / 2.0
    Ry = R[4] / 2.0
    Rz = R[5] / 2.0

    Cx = cos(Rx)
    Sx = sin(Rx)
    Cy = cos(Ry)
    Sy = sin(Ry)
    Cz = cos(Rz)
    Sz = sin(Rz)

    Angle = 2.0 * acos(Cx*Cy*Cz + Sx*Sy*Sz)
    x = Sx*Cy*Cz - Cx*Sy*Sz
    y = Cx*Sy*Cz + Sx*Cy*Sz
    z = -Sx*Sy*Cz + Cx*Cy*Sz
    Norm = sqrt(x*x + y*y + z*z)
    if norm(Norm) < 1e-4:
      Ax = 0
      Ay = 0
      Az = 0
    else:
    Ratio = Angle / Norm
    Ax = x * Ratio
    Ay = y * Ratio
    Az = z * Ratio
    end
    Ans = p[R[0], R[1], R[2], Ax, Ay, Az]

    return Ans
  end

  # Conversion (AxisAngle to RPY)
  def AxisAngle_to_RPY(R):
    Rx = R[3]
    Ry = R[4]
    Rz = R[5]

    Angle = sqrt(Rx*Rx + Ry*Ry + Rz*Rz)
    if Angle < 1e-4:
      x = 0
      y = 0
      z = 1
    else:
    x = Rx / Angle
    y = Ry / Angle
    z = Rz / Angle
    end
    S = sin(Angle)
    C = cos(Angle)
    T = 1 - C

    r11 = T*x*x + C
    r12 = T*x*y - S*z
    r13 = T*x*z + S*y
    r21 = T*x*y + S*z
    r22 = T*y*y + C
    r23 = T*y*z - S*x
    r31 = T*x*z - S*y
    r32 = T*y*z + S*x
    r33 = T*z*z + C

    if r31 > 1:
      r31 = 1
    elif r31 < -1:
      r31 = -1
    end

    Ay = asin(-r31)
    if Ay > d2r(89.9):
      sinAxMinusAz = (r12 - r23) / (1 - r31)
      cosAxMinusAz = (r13 + r22) / (1 - r31)
      Ax = atan2(sinAxMinusAz, cosAxMinusAz)
      Az =0
    elif Ay < d2r(-89.9):
      sinAxPlusAz = (-r12 - r23) / (1 + r31)
      cosAxPlusAz = (-r13 + r22) / (1 + r31)
      Ax = atan2(sinAxPlusAz, cosAxPlusAz)
      Az = 0
    else:
      Ax = atan2(r32, r33)
      Az = atan2(r21, r11)
    end

    Ans = p[R[0], R[1], R[2], Ax, Ay, Az]

    return Ans
  end

  # Get position in RPY coordinate
  def get_actual_tcp_pose_RPY():
    R = get_actual_tcp_pose()
    A = AxisAngle_to_RPY(R)

    return A
  end

  # Add position
  def pose_add_RPY(V1, V2):
    A0 = V1[0] + V2[0]
    A1 = V1[1] + V2[1]
    A2 = V1[2] + V2[2]
    A3 = V1[3] + V2[3]
    A4 = V1[4] + V2[4]
    A5 = V1[5] + V2[5]
    A = p[A0, A1, A2, A3, A4, A5]

    return A
  end
  $ 3 "CUR_SetUpCamera('Cam1', '192.168.0.10', 8500)"
  CUR_SetUpCamera("Cam1", "192.168.0.10", 8500)
  $ 4 "If CUR_InitComm('Cam1')==False"
  if (CUR_InitComm("Cam1")==False):
    $ 5 "Popup: Communication Lost"
    popup("Communication Lost", "Message", False, False, blocking=True)
  end
  while (True):
    $ 6 "Robot Program"
    $ 7 "Loop"
    while (True):
      $ 8 "triggerResult≔CUR_ProcCommand('Cam1')"
      global triggerResult=CUR_ProcCommand("Cam1")
      $ 9 "If triggerResult==1"
      if (triggerResult==1):
      end
    end
    $ 11 "CUR_CloseComm('Cam1')"
    CUR_CloseComm("Cam1")
    $ 12 "Halt"
    halt
  end
end
